KUKA KRL program: f1_Kuka_APT210T03S10.SRC

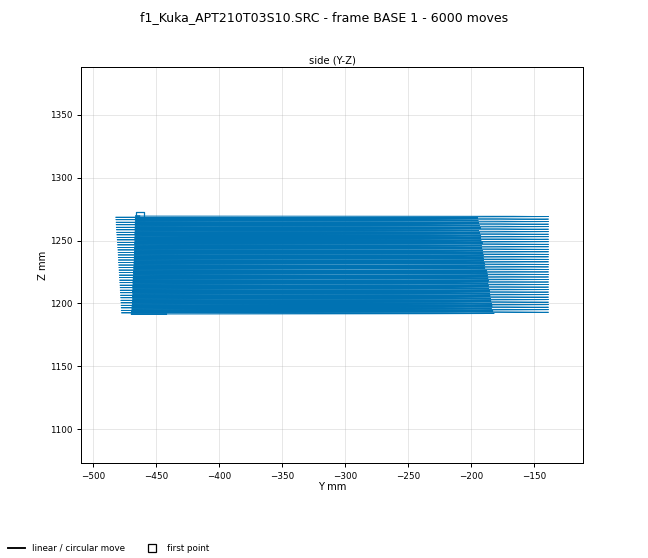
[picture p0: tool path of f1_Kuka_APT210T03S10.SRC in frame BASE 1, 6000 of 6001 moves have a stored position in this frame; points joined in program order, loops and branches not executed]
&ACCESS RVP
&REL 2
&PARAM TEMPLATE = C:\KRC\Roboter\Template\vorgabe
&PARAM EDITMASK = *
DEF f1_Kuka_APT210T03S10()


;FOLD INI;%{PE}%V3.2.0,%MKUKATPBASIS,%CINIT,%VCOMMON,%P
  ;FOLD BAS INI;%{E}%V3.2.0,%MKUKATPBASIS,%CINIT,%VINIT,%P
    GLOBAL INTERRUPT DECL 3 WHEN $STOPMESS==TRUE DO IR_STOPM ( )
    INTERRUPT ON 3
    BAS (#INITMOV,0 )
  ;ENDFOLD (BAS INI)
  ;FOLD USER INI;%{E}%V3.2.0,%MKUKATPUSER,%CINIT,%VINIT,%P
    ;Make your modifications here
  ;ENDFOLD (USER INI)
;ENDFOLD (INI)


;*** Make Null PTP Move
  PTP $pos_act

;*** Auto Load The Correct TOOL Data
  $tool=tool_data[3]

;*** Auto Load The Correct BASE Data
  $base=base_data[1]

  $ADVANCE = 5

;*** Restate Last Velocity
MMPM(30000.0)
SetRPM(6000)
LIN {X 0.158,Y -463.021,Z 1269.560,A 0.000,B 0.000,C 90.000,E1 280.725} C_DIS
LIN {X -0.171,Y -464.425,Z 1269.557,A 0.000,B 0.000,C 90.000,E1 280.254} C_DIS
LIN {X -0.038,Y -465.530,Z 1269.554,A 0.000,B 0.000,C 90.000,E1 279.726} C_DIS
LIN {X 0.024,Y -466.258,Z 1269.551,A 0.000,B 0.000,C 90.000,E1 279.208} C_DIS
LIN {X 0.098,Y -466.685,Z 1269.548,A 0.000,B 0.000,C 90.000,E1 278.690} C_DIS
LIN {X 0.243,Y -466.710,Z 1269.546,A 0.000,B 0.000,C 90.000,E1 278.163} C_DIS
LIN {X -0.138,Y -466.297,Z 1269.543,A 0.000,B 0.000,C 90.000,E1 277.701} C_DIS
LIN {X -0.055,Y -465.423,Z 1269.540,A 0.000,B 0.000,C 90.000,E1 277.182} C_DIS
LIN {X 0.026,Y -464.151,Z 1269.537,A 0.000,B 0.000,C 90.000,E1 276.663} C_DIS
LIN {X 0.102,Y -462.450,Z 1269.534,A 0.000,B 0.000,C 90.000,E1 276.144} C_DIS
LIN {X -0.010,Y -459.279,Z 1269.530,A 0.000,B 0.000,C 90.000,E1 275.391} C_DIS
LIN {X -0.004,Y -456.730,Z 1269.527,A 0.000,B 0.000,C 90.000,E1 274.878} C_DIS
LIN {X 0.028,Y -453.616,Z 1269.524,A 0.000,B 0.000,C 90.000,E1 274.359} C_DIS
LIN {X -0.204,Y -451.853,Z 1269.523,A 0.000,B 0.000,C 90.000,E1 274.131} C_DIS
LIN {X 0.039,Y -449.773,Z 1269.521,A 0.000,B 0.000,C 90.000,E1 273.841} C_DIS
LIN {X 0.001,Y -444.794,Z 1269.518,A 0.000,B 0.000,C 90.000,E1 273.326} C_DIS
LIN {X -0.204,Y -438.833,Z 1269.516,A 0.000,B 0.000,C 90.000,E1 272.865} C_DIS
LIN {X 0.074,Y -432.298,Z 1269.513,A 0.000,B 0.000,C 90.000,E1 272.407} C_DIS
LIN {X -0.016,Y -425.467,Z 1269.511,A 0.000,B 0.000,C 90.000,E1 272.064} C_DIS
LIN {X -0.063,Y -418.581,Z 1269.510,A 0.000,B 0.000,C 90.000,E1 271.776} C_DIS
LIN {X -0.186,Y -411.540,Z 1269.508,A 0.000,B 0.000,C 90.000,E1 271.547} C_DIS
LIN {X -0.025,Y -404.479,Z 1269.507,A 0.000,B 0.000,C 90.000,E1 271.318} C_DIS
LIN {X -0.034,Y -397.370,Z 1269.506,A 0.000,B 0.000,C 90.000,E1 271.146} C_DIS
LIN {X 0.152,Y -389.939,Z 1269.505,A 0.000,B 0.000,C 90.000,E1 270.974} C_DIS
LIN {X 0.139,Y -381.517,Z 1269.505,A 0.000,B 0.000,C 90.000,E1 270.859} C_DIS
LIN {X 0.169,Y -367.307,Z 1269.504,A 0.000,B 0.000,C 90.000,E1 270.745} C_DIS
LIN {X 0.045,Y -359.990,Z 1269.504,A 0.000,B 0.000,C 90.000,E1 270.745} C_DIS
LIN {X -0.008,Y -181.516,Z 1269.504,A 0.000,B 0.000,C 90.000,E1 270.745} C_DIS
LIN {X -0.022,Y -181.492,Z 1269.498,A 0.000,B 0.000,C 90.000,E1 269.714} C_DIS
LIN {X -0.079,Y -180.906,Z 1269.474,A 0.000,B 0.000,C 90.000,E1 265.355} C_DIS
LIN {X -0.005,Y -180.669,Z 1269.469,A 0.000,B 0.000,C 90.000,E1 264.489} C_DIS
LIN {X 0.070,Y -178.750,Z 1269.441,A 0.000,B 0.000,C 90.000,E1 259.398} C_DIS
LIN {X -0.033,Y -175.797,Z 1269.413,A 0.000,B 0.000,C 90.000,E1 254.338} C_DIS
LIN {X -0.038,Y -171.983,Z 1269.384,A 0.000,B 0.000,C 90.000,E1 249.209} C_DIS
LIN {X -0.001,Y -171.388,Z 1269.380,A 0.000,B 0.000,C 90.000,E1 248.337} C_DIS
LIN {X -0.015,Y -167.632,Z 1269.356,A 0.000,B 0.000,C 90.000,E1 244.024} C_DIS
LIN {X 0.000,Y -166.289,Z 1269.346,A 0.000,B 0.000,C 90.000,E1 242.281} C_DIS
LIN {X -0.006,Y -163.036,Z 1269.327,A 0.000,B 0.000,C 90.000,E1 238.791} C_DIS
LIN {X -0.044,Y -160.966,Z 1269.312,A 0.000,B 0.000,C 90.000,E1 236.167} C_DIS
LIN {X -0.066,Y -157.719,Z 1269.292,A 0.000,B 0.000,C 90.000,E1 232.637} C_DIS
LIN {X 0.092,Y -155.759,Z 1269.277,A 0.000,B 0.000,C 90.000,E1 229.908} C_DIS
LIN {X -0.071,Y -152.014,Z 1269.253,A 0.000,B 0.000,C 90.000,E1 225.486} C_DIS
LIN {X -0.053,Y -150.261,Z 1269.238,A 0.000,B 0.000,C 90.000,E1 222.771} C_DIS
LIN {X -0.034,Y -147.015,Z 1269.212,A 0.000,B 0.000,C 90.000,E1 218.222} C_DIS
LIN {X -0.013,Y -145.598,Z 1269.197,A 0.000,B 0.000,C 90.000,E1 215.471} C_DIS
LIN {X -0.009,Y -142.984,Z 1269.172,A 0.000,B 0.000,C 90.000,E1 210.875} C_DIS
LIN {X -0.009,Y -141.612,Z 1269.151,A 0.000,B 0.000,C 90.000,E1 207.180} C_DIS
LIN {X 0.032,Y -139.428,Z 1269.115,A 0.000,B 0.000,C 90.000,E1 200.663} C_DIS
LIN {X 0.083,Y -139.157,Z 1269.104,A 0.000,B 0.000,C 90.000,E1 198.779} C_DIS
LIN {X -0.031,Y -138.343,Z 1269.058,A 0.000,B 0.000,C 90.000,E1 190.423} C_DIS
LIN {X -0.049,Y -139.481,Z 1269.006,A 0.000,B 0.000,C 90.000,E1 181.088} C_DIS
LIN {X 0.031,Y -141.073,Z 1268.975,A 0.000,B 0.000,C 90.000,E1 175.469} C_DIS
LIN {X -0.014,Y -142.449,Z 1268.959,A 0.000,B 0.000,C 90.000,E1 172.704} C_DIS
LIN {X 0.076,Y -144.690,Z 1268.934,A 0.000,B 0.000,C 90.000,E1 168.049} C_DIS
LIN {X 0.028,Y -147.283,Z 1268.913,A 0.000,B 0.000,C 90.000,E1 164.393} C_DIS
LIN {X 0.045,Y -150.601,Z 1268.888,A 0.000,B 0.000,C 90.000,E1 159.826} C_DIS
LIN {X -0.019,Y -154.074,Z 1268.868,A 0.000,B 0.000,C 90.000,E1 156.230} C_DIS
LIN {X 0.047,Y -157.495,Z 1268.848,A 0.000,B 0.000,C 90.000,E1 152.615} C_DIS
LIN {X -0.008,Y -161.723,Z 1268.828,A 0.000,B 0.000,C 90.000,E1 149.076} C_DIS
LIN {X 0.006,Y -165.916,Z 1268.809,A 0.000,B 0.000,C 90.000,E1 145.548} C_DIS
LIN {X -0.008,Y -170.902,Z 1268.789,A 0.000,B 0.000,C 90.000,E1 142.065} C_DIS
LIN {X 0.019,Y -175.771,Z 1268.770,A 0.000,B 0.000,C 90.000,E1 138.609} C_DIS
LIN {X 0.020,Y -181.380,Z 1268.751,A 0.000,B 0.000,C 90.000,E1 135.202} C_DIS
LIN {X 0.025,Y -186.876,Z 1268.732,A 0.000,B 0.000,C 90.000,E1 131.838} C_DIS
LIN {X -0.023,Y -191.460,Z 1268.719,A 0.000,B 0.000,C 90.000,E1 129.358} C_DIS
LIN {X -0.091,Y -197.316,Z 1268.700,A 0.000,B 0.000,C 90.000,E1 126.091} C_DIS
LIN {X 0.035,Y -200.055,Z 1268.693,A 0.000,B 0.000,C 90.000,E1 124.692} C_DIS
LIN {X 0.012,Y -310.049,Z 1268.693,A 0.000,B 0.000,C 90.000,E1 124.692} C_DIS
LIN {X -0.114,Y -311.370,Z 1268.693,A 0.000,B 0.000,C 90.000,E1 124.692} C_DIS
LIN {X 0.173,Y -316.311,Z 1268.691,A 0.000,B 0.000,C 90.000,E1 124.405} C_DIS
LIN {X 0.136,Y -319.511,Z 1268.690,A 0.000,B 0.000,C 90.000,E1 124.119} C_DIS
LIN {X -0.031,Y -323.137,Z 1268.687,A 0.000,B 0.000,C 90.000,E1 123.627} C_DIS
LIN {X 0.048,Y -324.685,Z 1268.685,A 0.000,B 0.000,C 90.000,E1 123.293} C_DIS
LIN {X -0.059,Y -338.983,Z 1268.664,A 0.000,B 0.000,C 90.000,E1 119.539} C_DIS
LIN {X 0.108,Y -351.212,Z 1268.649,A 0.000,B 0.000,C 90.000,E1 116.744} C_DIS
LIN {X -0.164,Y -364.920,Z 1268.634,A 0.000,B 0.000,C 90.000,E1 114.079} C_DIS
LIN {X -0.132,Y -378.444,Z 1268.620,A 0.000,B 0.000,C 90.000,E1 111.716} C_DIS
LIN {X -0.031,Y -393.330,Z 1268.608,A 0.000,B 0.000,C 90.000,E1 109.396} C_DIS
LIN {X -0.067,Y -409.679,Z 1268.595,A 0.000,B 0.000,C 90.000,E1 107.149} C_DIS
LIN {X -0.068,Y -427.608,Z 1268.583,A 0.000,B 0.000,C 90.000,E1 104.954} C_DIS
LIN {X -0.038,Y -447.106,Z 1268.571,A 0.000,B 0.000,C 90.000,E1 102.827} C_DIS
LIN {X 0.166,Y -467.351,Z 1268.560,A 0.000,B 0.000,C 90.000,E1 100.838} C_DIS
LIN {X 0.180,Y -475.077,Z 1268.557,A 0.000,B 0.000,C 90.000,E1 100.141} C_DIS
LIN {X 0.231,Y -477.182,Z 1268.555,A 0.000,B 0.000,C 90.000,E1 99.905} C_DIS
LIN {X -0.191,Y -478.780,Z 1268.554,A 0.000,B 0.000,C 90.000,E1 99.726} C_DIS
LIN {X 0.075,Y -480.108,Z 1268.552,A 0.000,B 0.000,C 90.000,E1 99.443} C_DIS
LIN {X -0.053,Y -481.089,Z 1268.551,A 0.000,B 0.000,C 90.000,E1 99.208} C_DIS
LIN {X 0.108,Y -482.190,Z 1268.548,A 0.000,B 0.000,C 90.000,E1 98.690} C_DIS
LIN {X -0.131,Y -482.289,Z 1268.546,A 0.000,B 0.000,C 90.000,E1 98.219} C_DIS
LIN {X 0.042,Y -481.405,Z 1268.543,A 0.000,B 0.000,C 90.000,E1 97.701} C_DIS
LIN {X 0.217,Y -479.386,Z 1268.540,A 0.000,B 0.000,C 90.000,E1 97.182} C_DIS
LIN {X 0.093,Y -477.822,Z 1268.539,A 0.000,B 0.000,C 90.000,E1 96.947} C_DIS
LIN {X -0.096,Y -461.310,Z 1268.526,A 0.000,B 0.000,C 90.000,E1 94.702} C_DIS
LIN {X 0.147,Y -445.618,Z 1268.513,A 0.000,B 0.000,C 90.000,E1 92.350} C_DIS
LIN {X -0.178,Y -432.570,Z 1268.501,A 0.000,B 0.000,C 90.000,E1 90.286} C_DIS
LIN {X 0.076,Y -414.803,Z 1268.484,A 0.000,B 0.000,C 90.000,E1 87.020} C_DIS
LIN {X -0.112,Y -404.774,Z 1268.473,A 0.000,B 0.000,C 90.000,E1 85.122} C_DIS
LIN {X -0.122,Y -396.062,Z 1268.464,A 0.000,B 0.000,C 90.000,E1 83.451} C_DIS
LIN {X 0.134,Y -385.703,Z 1268.453,A 0.000,B 0.000,C 90.000,E1 81.432} C_DIS
LIN {X -0.114,Y -376.640,Z 1268.443,A 0.000,B 0.000,C 90.000,E1 79.746} C_DIS
LIN {X -0.080,Y -367.188,Z 1268.433,A 0.000,B 0.000,C 90.000,E1 77.993} C_DIS
LIN {X -0.100,Y -359.050,Z 1268.425,A 0.000,B 0.000,C 90.000,E1 76.520} C_DIS
LIN {X 0.054,Y -347.571,Z 1268.413,A 0.000,B 0.000,C 90.000,E1 74.393} C_DIS
LIN {X 0.032,Y -334.469,Z 1268.400,A 0.000,B 0.000,C 90.000,E1 71.945} C_DIS
LIN {X -0.036,Y -320.293,Z 1268.384,A 0.000,B 0.000,C 90.000,E1 69.135} C_DIS
LIN {X -0.150,Y -304.085,Z 1268.364,A 0.000,B 0.000,C 90.000,E1 65.613} C_DIS
LIN {X -0.020,Y -292.232,Z 1268.348,A 0.000,B 0.000,C 90.000,E1 62.615} C_DIS
LIN {X 0.106,Y -279.452,Z 1268.327,A 0.000,B 0.000,C 90.000,E1 58.869} C_DIS
LIN {X -0.065,Y -270.033,Z 1268.310,A 0.000,B 0.000,C 90.000,E1 55.801} C_DIS
LIN {X 0.025,Y -260.411,Z 1268.290,A 0.000,B 0.000,C 90.000,E1 52.271} C_DIS
LIN {X 0.015,Y -253.234,Z 1268.275,A 0.000,B 0.000,C 90.000,E1 49.417} C_DIS
LIN {X -0.068,Y -244.624,Z 1268.254,A 0.000,B 0.000,C 90.000,E1 45.810} C_DIS
LIN {X -0.071,Y -236.646,Z 1268.234,A 0.000,B 0.000,C 90.000,E1 42.123} C_DIS
LIN {X -0.096,Y -229.157,Z 1268.213,A 0.000,B 0.000,C 90.000,E1 38.382} C_DIS
LIN {X 0.083,Y -222.331,Z 1268.192,A 0.000,B 0.000,C 90.000,E1 34.532} C_DIS
LIN {X 0.099,Y -216.238,Z 1268.171,A 0.000,B 0.000,C 90.000,E1 30.669} C_DIS
LIN {X -0.029,Y -210.768,Z 1268.149,A 0.000,B 0.000,C 90.000,E1 26.796} C_DIS
LIN {X 0.046,Y -206.032,Z 1268.127,A 0.000,B 0.000,C 90.000,E1 22.823} C_DIS
LIN {X -0.048,Y -201.303,Z 1268.100,A 0.000,B 0.000,C 90.000,E1 18.055} C_DIS
LIN {X 0.084,Y -197.587,Z 1268.073,A 0.000,B 0.000,C 90.000,E1 13.175} C_DIS
LIN {X -0.088,Y -194.592,Z 1268.042,A 0.000,B 0.000,C 90.000,E1 7.530} C_DIS
LIN {X -0.068,Y -195.631,Z 1267.956,A 0.000,B 0.000,C 90.000,E1 352.186} C_DIS
LIN {X 0.023,Y -199.328,Z 1267.925,A 0.000,B 0.000,C 90.000,E1 346.464} C_DIS
LIN {X -0.029,Y -203.599,Z 1267.898,A 0.000,B 0.000,C 90.000,E1 341.638} C_DIS
LIN {X 0.062,Y -207.896,Z 1267.876,A 0.000,B 0.000,C 90.000,E1 337.614} C_DIS
LIN {X 0.115,Y -212.948,Z 1267.854,A 0.000,B 0.000,C 90.000,E1 333.640} C_DIS
LIN {X 0.043,Y -218.627,Z 1267.832,A 0.000,B 0.000,C 90.000,E1 329.744} C_DIS
LIN {X 0.023,Y -225.096,Z 1267.810,A 0.000,B 0.000,C 90.000,E1 325.881} C_DIS
LIN {X 0.029,Y -232.402,Z 1267.789,A 0.000,B 0.000,C 90.000,E1 322.065} C_DIS
LIN {X -0.034,Y -240.571,Z 1267.768,A 0.000,B 0.000,C 90.000,E1 318.324} C_DIS
LIN {X 0.122,Y -249.787,Z 1267.748,A 0.000,B 0.000,C 90.000,E1 314.595} C_DIS
LIN {X 0.007,Y -257.116,Z 1267.734,A 0.000,B 0.000,C 90.000,E1 312.081} C_DIS
LIN {X 0.077,Y -265.464,Z 1267.720,A 0.000,B 0.000,C 90.000,E1 309.564} C_DIS
LIN {X 0.122,Y -273.667,Z 1267.708,A 0.000,B 0.000,C 90.000,E1 307.443} C_DIS
LIN {X -0.005,Y -282.937,Z 1267.697,A 0.000,B 0.000,C 90.000,E1 305.391} C_DIS
LIN {X -0.123,Y -293.218,Z 1267.685,A 0.000,B 0.000,C 90.000,E1 303.372} C_DIS
LIN {X 0.028,Y -302.560,Z 1267.676,A 0.000,B 0.000,C 90.000,E1 301.671} C_DIS
LIN {X 0.134,Y -310.858,Z 1267.669,A 0.000,B 0.000,C 90.000,E1 300.335} C_DIS
LIN {X -0.082,Y -319.939,Z 1267.661,A 0.000,B 0.000,C 90.000,E1 299.077} C_DIS
LIN {X -0.060,Y -339.665,Z 1267.647,A 0.000,B 0.000,C 90.000,E1 296.539} C_DIS
LIN {X 0.032,Y -357.895,Z 1267.635,A 0.000,B 0.000,C 90.000,E1 294.387} C_DIS
LIN {X 0.075,Y -370.867,Z 1267.627,A 0.000,B 0.000,C 90.000,E1 292.898} C_DIS
LIN {X -0.027,Y -383.639,Z 1267.619,A 0.000,B 0.000,C 90.000,E1 291.461} C_DIS
LIN {X -0.057,Y -398.664,Z 1267.610,A 0.000,B 0.000,C 90.000,E1 289.758} C_DIS
LIN {X -0.116,Y -416.277,Z 1267.599,A 0.000,B 0.000,C 90.000,E1 287.873} C_DIS
LIN {X -0.219,Y -426.089,Z 1267.593,A 0.000,B 0.000,C 90.000,E1 286.804} C_DIS
LIN {X -0.040,Y -432.978,Z 1267.589,A 0.000,B 0.000,C 90.000,E1 285.969} C_DIS
LIN {X -0.210,Y -439.391,Z 1267.584,A 0.000,B 0.000,C 90.000,E1 285.190} C_DIS
LIN {X 0.092,Y -445.134,Z 1267.580,A 0.000,B 0.000,C 90.000,E1 284.356} C_DIS
LIN {X -0.088,Y -450.216,Z 1267.575,A 0.000,B 0.000,C 90.000,E1 283.592} C_DIS
LIN {X -0.229,Y -454.646,Z 1267.571,A 0.000,B 0.000,C 90.000,E1 282.827} C_DIS
LIN {X 0.120,Y -458.319,Z 1267.567,A 0.000,B 0.000,C 90.000,E1 282.007} C_DIS
LIN {X 0.052,Y -461.356,Z 1267.563,A 0.000,B 0.000,C 90.000,E1 281.243} C_DIS
LIN {X 0.079,Y -463.002,Z 1267.560,A 0.000,B 0.000,C 90.000,E1 280.725} C_DIS
LIN {X 0.206,Y -464.426,Z 1267.557,A 0.000,B 0.000,C 90.000,E1 280.197} C_DIS
LIN {X -0.119,Y -465.517,Z 1267.554,A 0.000,B 0.000,C 90.000,E1 279.726} C_DIS
LIN {X -0.057,Y -466.289,Z 1267.551,A 0.000,B 0.000,C 90.000,E1 279.208} C_DIS
LIN {X 0.087,Y -466.729,Z 1267.548,A 0.000,B 0.000,C 90.000,E1 278.681} C_DIS
LIN {X 0.163,Y -466.768,Z 1267.545,A 0.000,B 0.000,C 90.000,E1 278.163} C_DIS
LIN {X -0.218,Y -466.373,Z 1267.543,A 0.000,B 0.000,C 90.000,E1 277.701} C_DIS
LIN {X -0.135,Y -465.526,Z 1267.540,A 0.000,B 0.000,C 90.000,E1 277.182} C_DIS
LIN {X -0.053,Y -464.254,Z 1267.537,A 0.000,B 0.000,C 90.000,E1 276.663} C_DIS
LIN {X 0.023,Y -462.607,Z 1267.534,A 0.000,B 0.000,C 90.000,E1 276.144} C_DIS
LIN {X -0.086,Y -459.480,Z 1267.530,A 0.000,B 0.000,C 90.000,E1 275.391} C_DIS
LIN {X -0.078,Y -456.957,Z 1267.527,A 0.000,B 0.000,C 90.000,E1 274.878} C_DIS
LIN {X -0.046,Y -453.897,Z 1267.524,A 0.000,B 0.000,C 90.000,E1 274.359} C_DIS
LIN {X -0.033,Y -450.045,Z 1267.521,A 0.000,B 0.000,C 90.000,E1 273.841} C_DIS
LIN {X -0.068,Y -445.071,Z 1267.518,A 0.000,B 0.000,C 90.000,E1 273.326} C_DIS
LIN {X 0.140,Y -439.130,Z 1267.516,A 0.000,B 0.000,C 90.000,E1 272.808} C_DIS
LIN {X -0.049,Y -432.570,Z 1267.513,A 0.000,B 0.000,C 90.000,E1 272.407} C_DIS
LIN {X -0.148,Y -425.696,Z 1267.511,A 0.000,B 0.000,C 90.000,E1 272.064} C_DIS
LIN {X 0.202,Y -418.795,Z 1267.510,A 0.000,B 0.000,C 90.000,E1 271.718} C_DIS
LIN {X 0.061,Y -411.685,Z 1267.508,A 0.000,B 0.000,C 90.000,E1 271.489} C_DIS
LIN {X -0.045,Y -400.883,Z 1267.507,A 0.000,B 0.000,C 90.000,E1 271.203} C_DIS
LIN {X -0.026,Y -389.864,Z 1267.505,A 0.000,B 0.000,C 90.000,E1 270.974} C_DIS
LIN {X -0.034,Y -381.152,Z 1267.505,A 0.000,B 0.000,C 90.000,E1 270.859} C_DIS
LIN {X 0.002,Y -366.340,Z 1267.504,A 0.000,B 0.000,C 90.000,E1 270.745} C_DIS
LIN {X -0.060,Y -363.755,Z 1267.504,A 0.000,B 0.000,C 90.000,E1 270.745} C_DIS
LIN {X -0.062,Y -181.520,Z 1267.504,A 0.000,B 0.000,C 90.000,E1 270.745} C_DIS
LIN {X -0.014,Y -181.493,Z 1267.498,A 0.000,B 0.000,C 90.000,E1 269.714} C_DIS
LIN {X -0.071,Y -180.905,Z 1267.474,A 0.000,B 0.000,C 90.000,E1 265.355} C_DIS
LIN {X 0.003,Y -180.670,Z 1267.469,A 0.000,B 0.000,C 90.000,E1 264.489} C_DIS
LIN {X 0.077,Y -178.751,Z 1267.441,A 0.000,B 0.000,C 90.000,E1 259.398} C_DIS
LIN {X -0.026,Y -175.799,Z 1267.413,A 0.000,B 0.000,C 90.000,E1 254.338} C_DIS
LIN {X -0.030,Y -171.984,Z 1267.384,A 0.000,B 0.000,C 90.000,E1 249.209} C_DIS
LIN {X 0.008,Y -171.390,Z 1267.380,A 0.000,B 0.000,C 90.000,E1 248.337} C_DIS
LIN {X -0.008,Y -167.634,Z 1267.356,A 0.000,B 0.000,C 90.000,E1 244.024} C_DIS
LIN {X 0.008,Y -166.291,Z 1267.346,A 0.000,B 0.000,C 90.000,E1 242.281} C_DIS
LIN {X 0.002,Y -163.038,Z 1267.327,A 0.000,B 0.000,C 90.000,E1 238.791} C_DIS
LIN {X -0.037,Y -160.969,Z 1267.312,A 0.000,B 0.000,C 90.000,E1 236.167} C_DIS
LIN {X -0.059,Y -157.721,Z 1267.292,A 0.000,B 0.000,C 90.000,E1 232.637} C_DIS
LIN {X 0.100,Y -155.760,Z 1267.277,A 0.000,B 0.000,C 90.000,E1 229.908} C_DIS
LIN {X -0.063,Y -152.017,Z 1267.253,A 0.000,B 0.000,C 90.000,E1 225.486} C_DIS
LIN {X -0.045,Y -150.263,Z 1267.238,A 0.000,B 0.000,C 90.000,E1 222.771} C_DIS
LIN {X -0.027,Y -147.017,Z 1267.212,A 0.000,B 0.000,C 90.000,E1 218.222} C_DIS
LIN {X -0.006,Y -145.599,Z 1267.197,A 0.000,B 0.000,C 90.000,E1 215.471} C_DIS
LIN {X -0.002,Y -142.986,Z 1267.172,A 0.000,B 0.000,C 90.000,E1 210.875} C_DIS
LIN {X -0.002,Y -141.613,Z 1267.151,A 0.000,B 0.000,C 90.000,E1 207.180} C_DIS
LIN {X 0.039,Y -139.428,Z 1267.115,A 0.000,B 0.000,C 90.000,E1 200.663} C_DIS
LIN {X -0.042,Y -139.158,Z 1267.104,A 0.000,B 0.000,C 90.000,E1 198.833} C_DIS
LIN {X -0.024,Y -138.342,Z 1267.058,A 0.000,B 0.000,C 90.000,E1 190.423} C_DIS
LIN {X -0.042,Y -139.481,Z 1267.006,A 0.000,B 0.000,C 90.000,E1 181.088} C_DIS
LIN {X 0.039,Y -141.073,Z 1266.975,A 0.000,B 0.000,C 90.000,E1 175.469} C_DIS
LIN {X -0.007,Y -142.448,Z 1266.959,A 0.000,B 0.000,C 90.000,E1 172.704} C_DIS
LIN {X 0.083,Y -144.689,Z 1266.934,A 0.000,B 0.000,C 90.000,E1 168.049} C_DIS
LIN {X 0.036,Y -147.281,Z 1266.913,A 0.000,B 0.000,C 90.000,E1 164.393} C_DIS
LIN {X 0.052,Y -150.599,Z 1266.888,A 0.000,B 0.000,C 90.000,E1 159.826} C_DIS
LIN {X -0.012,Y -154.072,Z 1266.868,A 0.000,B 0.000,C 90.000,E1 156.230} C_DIS
LIN {X 0.054,Y -157.492,Z 1266.848,A 0.000,B 0.000,C 90.000,E1 152.615} C_DIS
LIN {X 0.000,Y -161.719,Z 1266.828,A 0.000,B 0.000,C 90.000,E1 149.076} C_DIS
LIN {X 0.013,Y -165.913,Z 1266.809,A 0.000,B 0.000,C 90.000,E1 145.548} C_DIS
LIN {X 0.001,Y -170.899,Z 1266.789,A 0.000,B 0.000,C 90.000,E1 142.065} C_DIS
LIN {X 0.028,Y -175.767,Z 1266.770,A 0.000,B 0.000,C 90.000,E1 138.609} C_DIS
LIN {X -0.100,Y -181.376,Z 1266.751,A 0.000,B 0.000,C 90.000,E1 135.243} C_DIS
LIN {X 0.033,Y -186.871,Z 1266.733,A 0.000,B 0.000,C 90.000,E1 131.838} C_DIS
LIN {X -0.014,Y -191.455,Z 1266.719,A 0.000,B 0.000,C 90.000,E1 129.358} C_DIS
LIN {X -0.082,Y -197.310,Z 1266.700,A 0.000,B 0.000,C 90.000,E1 126.091} C_DIS
LIN {X -0.012,Y -200.083,Z 1266.693,A 0.000,B 0.000,C 90.000,E1 124.692} C_DIS
LIN {X -0.061,Y -309.766,Z 1266.693,A 0.000,B 0.000,C 90.000,E1 124.692} C_DIS
LIN {X -0.073,Y -316.076,Z 1266.691,A 0.000,B 0.000,C 90.000,E1 124.452} C_DIS
LIN {X -0.096,Y -319.047,Z 1266.690,A 0.000,B 0.000,C 90.000,E1 124.199} C_DIS
LIN {X -0.141,Y -322.741,Z 1266.687,A 0.000,B 0.000,C 90.000,E1 123.706} C_DIS
LIN {X -0.063,Y -324.386,Z 1266.685,A 0.000,B 0.000,C 90.000,E1 123.372} C_DIS
LIN {X -0.062,Y -327.900,Z 1266.680,A 0.000,B 0.000,C 90.000,E1 122.418} C_DIS
LIN {X -0.010,Y -338.723,Z 1266.664,A 0.000,B 0.000,C 90.000,E1 119.589} C_DIS
LIN {X -0.016,Y -350.922,Z 1266.649,A 0.000,B 0.000,C 90.000,E1 116.821} C_DIS
LIN {X 0.189,Y -364.596,Z 1266.634,A 0.000,B 0.000,C 90.000,E1 114.079} C_DIS
LIN {X -0.125,Y -378.092,Z 1266.621,A 0.000,B 0.000,C 90.000,E1 111.770} C_DIS
LIN {X -0.039,Y -392.943,Z 1266.608,A 0.000,B 0.000,C 90.000,E1 109.450} C_DIS
LIN {X -0.212,Y -409.258,Z 1266.595,A 0.000,B 0.000,C 90.000,E1 107.221} C_DIS
LIN {X -0.107,Y -427.148,Z 1266.583,A 0.000,B 0.000,C 90.000,E1 105.009} C_DIS
LIN {X -0.102,Y -446.616,Z 1266.572,A 0.000,B 0.000,C 90.000,E1 102.883} C_DIS
LIN {X 0.063,Y -466.847,Z 1266.561,A 0.000,B 0.000,C 90.000,E1 100.894} C_DIS
LIN {X 0.062,Y -474.584,Z 1266.557,A 0.000,B 0.000,C 90.000,E1 100.197} C_DIS
LIN {X 0.117,Y -476.776,Z 1266.555,A 0.000,B 0.000,C 90.000,E1 99.962} C_DIS
LIN {X 0.170,Y -478.434,Z 1266.554,A 0.000,B 0.000,C 90.000,E1 99.726} C_DIS
LIN {X -0.038,Y -479.815,Z 1266.553,A 0.000,B 0.000,C 90.000,E1 99.500} C_DIS
LIN {X -0.167,Y -480.839,Z 1266.551,A 0.000,B 0.000,C 90.000,E1 99.265} C_DIS
LIN {X -0.010,Y -482.013,Z 1266.549,A 0.000,B 0.000,C 90.000,E1 98.746} C_DIS
LIN {X 0.227,Y -482.176,Z 1266.546,A 0.000,B 0.000,C 90.000,E1 98.219} C_DIS
LIN {X -0.078,Y -481.361,Z 1266.543,A 0.000,B 0.000,C 90.000,E1 97.757} C_DIS
LIN {X 0.095,Y -479.428,Z 1266.540,A 0.000,B 0.000,C 90.000,E1 97.239} C_DIS
LIN {X -0.029,Y -477.924,Z 1266.539,A 0.000,B 0.000,C 90.000,E1 97.004} C_DIS
LIN {X 0.029,Y -459.641,Z 1266.525,A 0.000,B 0.000,C 90.000,E1 94.473} C_DIS
LIN {X -0.209,Y -444.016,Z 1266.512,A 0.000,B 0.000,C 90.000,E1 92.178} C_DIS
LIN {X 0.149,Y -432.605,Z 1266.502,A 0.000,B 0.000,C 90.000,E1 90.286} C_DIS
LIN {X -0.120,Y -416.277,Z 1266.485,A 0.000,B 0.000,C 90.000,E1 87.364} C_DIS
LIN {X 0.196,Y -404.829,Z 1266.473,A 0.000,B 0.000,C 90.000,E1 85.122} C_DIS
LIN {X 0.135,Y -396.116,Z 1266.464,A 0.000,B 0.000,C 90.000,E1 83.457} C_DIS
LIN {X 0.048,Y -385.759,Z 1266.453,A 0.000,B 0.000,C 90.000,E1 81.489} C_DIS
LIN {X 0.175,Y -376.705,Z 1266.443,A 0.000,B 0.000,C 90.000,E1 79.746} C_DIS
LIN {X -0.157,Y -367.282,Z 1266.433,A 0.000,B 0.000,C 90.000,E1 78.049} C_DIS
LIN {X 0.138,Y -357.506,Z 1266.424,A 0.000,B 0.000,C 90.000,E1 76.228} C_DIS
LIN {X -0.080,Y -346.034,Z 1266.412,A 0.000,B 0.000,C 90.000,E1 74.157} C_DIS
LIN {X -0.033,Y -332.990,Z 1266.398,A 0.000,B 0.000,C 90.000,E1 71.692} C_DIS
LIN {X 0.050,Y -318.884,Z 1266.383,A 0.000,B 0.000,C 90.000,E1 68.847} C_DIS
LIN {X -0.002,Y -302.828,Z 1266.363,A 0.000,B 0.000,C 90.000,E1 65.305} C_DIS
LIN {X -0.179,Y -291.108,Z 1266.346,A 0.000,B 0.000,C 90.000,E1 62.359} C_DIS
LIN {X -0.083,Y -278.399,Z 1266.326,A 0.000,B 0.000,C 90.000,E1 58.614} C_DIS
LIN {X 0.018,Y -268.019,Z 1266.306,A 0.000,B 0.000,C 90.000,E1 55.135} C_DIS
LIN {X -0.015,Y -258.521,Z 1266.287,A 0.000,B 0.000,C 90.000,E1 51.618} C_DIS
LIN {X -0.101,Y -251.379,Z 1266.271,A 0.000,B 0.000,C 90.000,E1 48.771} C_DIS
LIN {X 0.115,Y -242.871,Z 1266.251,A 0.000,B 0.000,C 90.000,E1 45.081} C_DIS
LIN {X -0.040,Y -236.536,Z 1266.234,A 0.000,B 0.000,C 90.000,E1 42.162} C_DIS
LIN {X 0.084,Y -228.992,Z 1266.213,A 0.000,B 0.000,C 90.000,E1 38.382} C_DIS
LIN {X -0.056,Y -222.126,Z 1266.192,A 0.000,B 0.000,C 90.000,E1 34.612} C_DIS
LIN {X 0.071,Y -215.931,Z 1266.171,A 0.000,B 0.000,C 90.000,E1 30.718} C_DIS
LIN {X 0.021,Y -210.428,Z 1266.149,A 0.000,B 0.000,C 90.000,E1 26.821} C_DIS
LIN {X -0.092,Y -205.670,Z 1266.127,A 0.000,B 0.000,C 90.000,E1 22.898} C_DIS
LIN {X 0.067,Y -200.912,Z 1266.100,A 0.000,B 0.000,C 90.000,E1 18.055} C_DIS
LIN {X -0.055,Y -197.201,Z 1266.073,A 0.000,B 0.000,C 90.000,E1 13.244} C_DIS
LIN {X -0.008,Y -194.235,Z 1266.042,A 0.000,B 0.000,C 90.000,E1 7.530} C_DIS
LIN {X -0.081,Y -195.435,Z 1265.956,A 0.000,B 0.000,C 90.000,E1 352.186} C_DIS
LIN {X 0.001,Y -199.169,Z 1265.925,A 0.000,B 0.000,C 90.000,E1 346.464} C_DIS
LIN {X -0.057,Y -203.482,Z 1265.898,A 0.000,B 0.000,C 90.000,E1 341.638} C_DIS
LIN {X 0.031,Y -207.817,Z 1265.876,A 0.000,B 0.000,C 90.000,E1 337.614} C_DIS
LIN {X 0.080,Y -212.892,Z 1265.854,A 0.000,B 0.000,C 90.000,E1 333.640} C_DIS
LIN {X 0.005,Y -218.568,Z 1265.832,A 0.000,B 0.000,C 90.000,E1 329.744} C_DIS
LIN {X -0.018,Y -225.073,Z 1265.810,A 0.000,B 0.000,C 90.000,E1 325.881} C_DIS
LIN {X -0.014,Y -232.373,Z 1265.789,A 0.000,B 0.000,C 90.000,E1 322.065} C_DIS
LIN {X -0.080,Y -240.543,Z 1265.768,A 0.000,B 0.000,C 90.000,E1 318.324} C_DIS
LIN {X 0.073,Y -249.757,Z 1265.748,A 0.000,B 0.000,C 90.000,E1 314.595} C_DIS
LIN {X -0.043,Y -257.088,Z 1265.734,A 0.000,B 0.000,C 90.000,E1 312.081} C_DIS
LIN {X 0.025,Y -265.425,Z 1265.720,A 0.000,B 0.000,C 90.000,E1 309.564} C_DIS
LIN {X -0.010,Y -275.069,Z 1265.706,A 0.000,B 0.000,C 90.000,E1 307.111} C_DIS
LIN {X 0.055,Y -284.540,Z 1265.695,A 0.000,B 0.000,C 90.000,E1 305.025} C_DIS
LIN {X -0.035,Y -294.944,Z 1265.683,A 0.000,B 0.000,C 90.000,E1 303.007} C_DIS
LIN {X -0.023,Y -304.456,Z 1265.674,A 0.000,B 0.000,C 90.000,E1 301.337} C_DIS
LIN {X 0.159,Y -315.221,Z 1265.665,A 0.000,B 0.000,C 90.000,E1 299.667} C_DIS
LIN {X 0.069,Y -334.565,Z 1265.651,A 0.000,B 0.000,C 90.000,E1 297.129} C_DIS
LIN {X 0.034,Y -354.844,Z 1265.637,A 0.000,B 0.000,C 90.000,E1 294.719} C_DIS
LIN {X 0.152,Y -367.931,Z 1265.629,A 0.000,B 0.000,C 90.000,E1 293.206} C_DIS
LIN {X 0.015,Y -380.718,Z 1265.621,A 0.000,B 0.000,C 90.000,E1 291.770} C_DIS
LIN {X -0.028,Y -395.809,Z 1265.611,A 0.000,B 0.000,C 90.000,E1 290.066} C_DIS
LIN {X 0.040,Y -416.031,Z 1265.599,A 0.000,B 0.000,C 90.000,E1 287.873} C_DIS
LIN {X -0.053,Y -425.865,Z 1265.593,A 0.000,B 0.000,C 90.000,E1 286.804} C_DIS
LIN {X 0.125,Y -432.793,Z 1265.589,A 0.000,B 0.000,C 90.000,E1 285.969} C_DIS
LIN {X -0.044,Y -439.200,Z 1265.584,A 0.000,B 0.000,C 90.000,E1 285.190} C_DIS
LIN {X -0.172,Y -444.974,Z 1265.580,A 0.000,B 0.000,C 90.000,E1 284.411} C_DIS
LIN {X 0.080,Y -450.085,Z 1265.576,A 0.000,B 0.000,C 90.000,E1 283.592} C_DIS
LIN {X -0.061,Y -454.490,Z 1265.571,A 0.000,B 0.000,C 90.000,E1 282.827} C_DIS
LIN {X -0.160,Y -458.186,Z 1265.567,A 0.000,B 0.000,C 90.000,E1 282.063} C_DIS
LIN {X 0.219,Y -461.264,Z 1265.563,A 0.000,B 0.000,C 90.000,E1 281.243} C_DIS
LIN {X -0.209,Y -462.922,Z 1265.560,A 0.000,B 0.000,C 90.000,E1 280.782} C_DIS
LIN {X -0.084,Y -464.330,Z 1265.557,A 0.000,B 0.000,C 90.000,E1 280.254} C_DIS
LIN {X 0.048,Y -465.445,Z 1265.554,A 0.000,B 0.000,C 90.000,E1 279.726} C_DIS
LIN {X 0.111,Y -466.298,Z 1265.551,A 0.000,B 0.000,C 90.000,E1 279.208} C_DIS
LIN {X 0.183,Y -466.746,Z 1265.548,A 0.000,B 0.000,C 90.000,E1 278.690} C_DIS
LIN {X -0.132,Y -466.824,Z 1265.546,A 0.000,B 0.000,C 90.000,E1 278.219} C_DIS
LIN {X -0.051,Y -466.498,Z 1265.543,A 0.000,B 0.000,C 90.000,E1 277.701} C_DIS
LIN {X 0.032,Y -465.680,Z 1265.540,A 0.000,B 0.000,C 90.000,E1 277.182} C_DIS
LIN {X 0.114,Y -464.471,Z 1265.537,A 0.000,B 0.000,C 90.000,E1 276.663} C_DIS
LIN {X 0.191,Y -462.850,Z 1265.534,A 0.000,B 0.000,C 90.000,E1 276.144} C_DIS
LIN {X 0.082,Y -459.799,Z 1265.530,A 0.000,B 0.000,C 90.000,E1 275.391} C_DIS
LIN {X 0.091,Y -457.330,Z 1265.527,A 0.000,B 0.000,C 90.000,E1 274.878} C_DIS
LIN {X 0.123,Y -454.306,Z 1265.524,A 0.000,B 0.000,C 90.000,E1 274.359} C_DIS
LIN {X -0.106,Y -452.554,Z 1265.523,A 0.000,B 0.000,C 90.000,E1 274.131} C_DIS
LIN {X -0.098,Y -448.264,Z 1265.520,A 0.000,B 0.000,C 90.000,E1 273.612} C_DIS
LIN {X 0.103,Y -445.689,Z 1265.519,A 0.000,B 0.000,C 90.000,E1 273.326} C_DIS
LIN {X -0.156,Y -439.827,Z 1265.516,A 0.000,B 0.000,C 90.000,E1 272.865} C_DIS
LIN {X 0.046,Y -433.328,Z 1265.513,A 0.000,B 0.000,C 90.000,E1 272.407} C_DIS
LIN {X -0.097,Y -426.481,Z 1265.511,A 0.000,B 0.000,C 90.000,E1 272.064} C_DIS
LIN {X -0.199,Y -419.529,Z 1265.510,A 0.000,B 0.000,C 90.000,E1 271.776} C_DIS
LIN {X 0.055,Y -412.463,Z 1265.508,A 0.000,B 0.000,C 90.000,E1 271.489} C_DIS
LIN {X -0.100,Y -401.739,Z 1265.507,A 0.000,B 0.000,C 90.000,E1 271.203} C_DIS
LIN {X -0.087,Y -393.911,Z 1265.506,A 0.000,B 0.000,C 90.000,E1 271.031} C_DIS
LIN {X 0.174,Y -385.825,Z 1265.505,A 0.000,B 0.000,C 90.000,E1 270.859} C_DIS
LIN {X -0.135,Y -375.921,Z 1265.504,A 0.000,B 0.000,C 90.000,E1 270.802} C_DIS
LIN {X 0.152,Y -362.858,Z 1265.504,A 0.000,B 0.000,C 90.000,E1 270.688} C_DIS
LIN {X 0.044,Y -181.526,Z 1265.504,A 0.000,B 0.000,C 90.000,E1 270.688} C_DIS
LIN {X -0.090,Y -181.487,Z 1265.498,A 0.000,B 0.000,C 90.000,E1 269.714} C_DIS
LIN {X 0.034,Y -180.904,Z 1265.474,A 0.000,B 0.000,C 90.000,E1 265.298} C_DIS
LIN {X -0.016,Y -180.248,Z 1265.465,A 0.000,B 0.000,C 90.000,E1 263.628} C_DIS
LIN {X 0.002,Y -178.737,Z 1265.441,A 0.000,B 0.000,C 90.000,E1 259.398} C_DIS
LIN {X 0.069,Y -175.785,Z 1265.413,A 0.000,B 0.000,C 90.000,E1 254.283} C_DIS
LIN {X 0.056,Y -171.969,Z 1265.384,A 0.000,B 0.000,C 90.000,E1 249.156} C_DIS
LIN {X 0.094,Y -171.369,Z 1265.380,A 0.000,B 0.000,C 90.000,E1 248.284} C_DIS
LIN {X -0.080,Y -167.616,Z 1265.356,A 0.000,B 0.000,C 90.000,E1 244.024} C_DIS
LIN {X -0.065,Y -166.265,Z 1265.346,A 0.000,B 0.000,C 90.000,E1 242.281} C_DIS
LIN {X 0.070,Y -163.018,Z 1265.327,A 0.000,B 0.000,C 90.000,E1 238.742} C_DIS
LIN {X -0.017,Y -160.943,Z 1265.312,A 0.000,B 0.000,C 90.000,E1 236.135} C_DIS
LIN {X 0.093,Y -157.701,Z 1265.292,A 0.000,B 0.000,C 90.000,E1 232.557} C_DIS
LIN {X 0.031,Y -155.740,Z 1265.277,A 0.000,B 0.000,C 90.000,E1 229.908} C_DIS
LIN {X 0.084,Y -151.998,Z 1265.252,A 0.000,B 0.000,C 90.000,E1 225.405} C_DIS
LIN {X -0.010,Y -150.243,Z 1265.237,A 0.000,B 0.000,C 90.000,E1 222.732} C_DIS
LIN {X 0.022,Y -147.002,Z 1265.212,A 0.000,B 0.000,C 90.000,E1 218.177} C_DIS
LIN {X 0.012,Y -145.586,Z 1265.197,A 0.000,B 0.000,C 90.000,E1 215.438} C_DIS
LIN {X 0.006,Y -142.974,Z 1265.171,A 0.000,B 0.000,C 90.000,E1 210.846} C_DIS
LIN {X 0.059,Y -141.601,Z 1265.151,A 0.000,B 0.000,C 90.000,E1 207.129} C_DIS
LIN {X -0.026,Y -139.423,Z 1265.115,A 0.000,B 0.000,C 90.000,E1 200.663} C_DIS
LIN {X 0.026,Y -139.152,Z 1265.104,A 0.000,B 0.000,C 90.000,E1 198.779} C_DIS
LIN {X 0.048,Y -138.345,Z 1265.058,A 0.000,B 0.000,C 90.000,E1 190.366} C_DIS
LIN {X 0.033,Y -139.485,Z 1265.006,A 0.000,B 0.000,C 90.000,E1 181.031} C_DIS
LIN {X -0.026,Y -141.084,Z 1264.975,A 0.000,B 0.000,C 90.000,E1 175.469} C_DIS
LIN {X -0.073,Y -142.461,Z 1264.959,A 0.000,B 0.000,C 90.000,E1 172.704} C_DIS
LIN {X 0.017,Y -144.704,Z 1264.934,A 0.000,B 0.000,C 90.000,E1 168.049} C_DIS
LIN {X -0.032,Y -147.302,Z 1264.913,A 0.000,B 0.000,C 90.000,E1 164.393} C_DIS
LIN {X -0.016,Y -150.621,Z 1264.888,A 0.000,B 0.000,C 90.000,E1 159.826} C_DIS
LIN {X 0.060,Y -154.096,Z 1264.868,A 0.000,B 0.000,C 90.000,E1 156.177} C_DIS
LIN {X -0.016,Y -157.520,Z 1264.848,A 0.000,B 0.000,C 90.000,E1 152.615} C_DIS
LIN {X -0.071,Y -161.752,Z 1264.828,A 0.000,B 0.000,C 90.000,E1 149.076} C_DIS
LIN {X 0.034,Y -165.945,Z 1264.808,A 0.000,B 0.000,C 90.000,E1 145.515} C_DIS
LIN {X 0.032,Y -170.936,Z 1264.789,A 0.000,B 0.000,C 90.000,E1 142.029} C_DIS
LIN {X -0.048,Y -175.804,Z 1264.770,A 0.000,B 0.000,C 90.000,E1 138.609} C_DIS
LIN {X 0.080,Y -181.413,Z 1264.751,A 0.000,B 0.000,C 90.000,E1 135.162} C_DIS
LIN {X -0.045,Y -186.914,Z 1264.732,A 0.000,B 0.000,C 90.000,E1 131.838} C_DIS
LIN {X 0.028,Y -191.494,Z 1264.719,A 0.000,B 0.000,C 90.000,E1 129.322} C_DIS
LIN {X 0.114,Y -197.356,Z 1264.700,A 0.000,B 0.000,C 90.000,E1 126.011} C_DIS
LIN {X -0.065,Y -200.115,Z 1264.693,A 0.000,B 0.000,C 90.000,E1 124.692} C_DIS
LIN {X -0.143,Y -309.647,Z 1264.693,A 0.000,B 0.000,C 90.000,E1 124.692} C_DIS
LIN {X -0.051,Y -310.862,Z 1264.693,A 0.000,B 0.000,C 90.000,E1 124.659} C_DIS
LIN {X 0.060,Y -316.209,Z 1264.691,A 0.000,B 0.000,C 90.000,E1 124.405} C_DIS
LIN {X 0.141,Y -319.277,Z 1264.690,A 0.000,B 0.000,C 90.000,E1 124.119} C_DIS
LIN {X 0.052,Y -322.944,Z 1264.687,A 0.000,B 0.000,C 90.000,E1 123.627} C_DIS
LIN {X 0.132,Y -324.551,Z 1264.685,A 0.000,B 0.000,C 90.000,E1 123.293} C_DIS
LIN {X -0.040,Y -329.179,Z 1264.678,A 0.000,B 0.000,C 90.000,E1 122.054} C_DIS
LIN {X 0.163,Y -340.172,Z 1264.662,A 0.000,B 0.000,C 90.000,E1 119.205} C_DIS
LIN {X -0.101,Y -352.549,Z 1264.647,A 0.000,B 0.000,C 90.000,E1 116.488} C_DIS
LIN {X -0.014,Y -366.424,Z 1264.632,A 0.000,B 0.000,C 90.000,E1 113.770} C_DIS
LIN {X 0.064,Y -380.106,Z 1264.619,A 0.000,B 0.000,C 90.000,E1 111.408} C_DIS
LIN {X -0.160,Y -395.161,Z 1264.606,A 0.000,B 0.000,C 90.000,E1 109.141} C_DIS
LIN {X 0.106,Y -411.692,Z 1264.594,A 0.000,B 0.000,C 90.000,E1 106.858} C_DIS
LIN {X -0.244,Y -429.819,Z 1264.582,A 0.000,B 0.000,C 90.000,E1 104.717} C_DIS
LIN {X -0.115,Y -449.462,Z 1264.570,A 0.000,B 0.000,C 90.000,E1 102.591} C_DIS
LIN {X -0.213,Y -469.772,Z 1264.559,A 0.000,B 0.000,C 90.000,E1 100.658} C_DIS
LIN {X -0.213,Y -474.908,Z 1264.557,A 0.000,B 0.000,C 90.000,E1 100.197} C_DIS
LIN {X -0.169,Y -476.992,Z 1264.555,A 0.000,B 0.000,C 90.000,E1 99.962} C_DIS
LIN {X -0.125,Y -478.575,Z 1264.554,A 0.000,B 0.000,C 90.000,E1 99.726} C_DIS
LIN {X 0.141,Y -479.887,Z 1264.553,A 0.000,B 0.000,C 90.000,E1 99.443} C_DIS
LIN {X 0.013,Y -480.854,Z 1264.551,A 0.000,B 0.000,C 90.000,E1 99.208} C_DIS
LIN {X 0.172,Y -481.933,Z 1264.548,A 0.000,B 0.000,C 90.000,E1 98.690} C_DIS
LIN {X -0.069,Y -482.012,Z 1264.546,A 0.000,B 0.000,C 90.000,E1 98.219} C_DIS
LIN {X 0.104,Y -481.107,Z 1264.543,A 0.000,B 0.000,C 90.000,E1 97.701} C_DIS
LIN {X -0.199,Y -479.063,Z 1264.540,A 0.000,B 0.000,C 90.000,E1 97.239} C_DIS
LIN {X 0.151,Y -477.482,Z 1264.539,A 0.000,B 0.000,C 90.000,E1 96.947} C_DIS
LIN {X -0.048,Y -460.979,Z 1264.526,A 0.000,B 0.000,C 90.000,E1 94.702} C_DIS
LIN {X 0.185,Y -445.277,Z 1264.513,A 0.000,B 0.000,C 90.000,E1 92.350} C_DIS
LIN {X -0.149,Y -432.173,Z 1264.501,A 0.000,B 0.000,C 90.000,E1 90.286} C_DIS
LIN {X -0.004,Y -415.869,Z 1264.485,A 0.000,B 0.000,C 90.000,E1 87.306} C_DIS
LIN {X -0.104,Y -404.427,Z 1264.473,A 0.000,B 0.000,C 90.000,E1 85.122} C_DIS
LIN {X -0.100,Y -394.235,Z 1264.462,A 0.000,B 0.000,C 90.000,E1 83.166} C_DIS
LIN {X 0.170,Y -383.880,Z 1264.451,A 0.000,B 0.000,C 90.000,E1 81.141} C_DIS
LIN {X -0.109,Y -374.723,Z 1264.441,A 0.000,B 0.000,C 90.000,E1 79.454} C_DIS
LIN {X -0.099,Y -366.867,Z 1264.433,A 0.000,B 0.000,C 90.000,E1 77.993} C_DIS
LIN {X 0.184,Y -357.105,Z 1264.423,A 0.000,B 0.000,C 90.000,E1 76.172} C_DIS
LIN {X -0.046,Y -345.643,Z 1264.412,A 0.000,B 0.000,C 90.000,E1 74.102} C_DIS
LIN {X -0.014,Y -332.615,Z 1264.398,A 0.000,B 0.000,C 90.000,E1 71.638} C_DIS
LIN {X 0.167,Y -318.537,Z 1264.382,A 0.000,B 0.000,C 90.000,E1 68.773} C_DIS
LIN {X 0.108,Y -302.532,Z 1264.363,A 0.000,B 0.000,C 90.000,E1 65.229} C_DIS
LIN {X -0.074,Y -290.831,Z 1264.346,A 0.000,B 0.000,C 90.000,E1 62.281} C_DIS
LIN {X 0.015,Y -278.096,Z 1264.325,A 0.000,B 0.000,C 90.000,E1 58.535} C_DIS
LIN {X -0.112,Y -267.677,Z 1264.306,A 0.000,B 0.000,C 90.000,E1 55.102} C_DIS
LIN {X 0.063,Y -258.159,Z 1264.286,A 0.000,B 0.000,C 90.000,E1 51.537} C_DIS
LIN {X -0.033,Y -251.029,Z 1264.271,A 0.000,B 0.000,C 90.000,E1 48.690} C_DIS
LIN {X 0.001,Y -242.516,Z 1264.250,A 0.000,B 0.000,C 90.000,E1 45.040} C_DIS
LIN {X 0.006,Y -236.169,Z 1264.234,A 0.000,B 0.000,C 90.000,E1 42.081} C_DIS
LIN {X -0.026,Y -228.588,Z 1264.213,A 0.000,B 0.000,C 90.000,E1 38.338} C_DIS
LIN {X -0.041,Y -221.688,Z 1264.192,A 0.000,B 0.000,C 90.000,E1 34.532} C_DIS
LIN {X -0.042,Y -215.437,Z 1264.170,A 0.000,B 0.000,C 90.000,E1 30.669} C_DIS
LIN {X -0.003,Y -209.926,Z 1264.149,A 0.000,B 0.000,C 90.000,E1 26.744} C_DIS
LIN {X 0.051,Y -205.167,Z 1264.127,A 0.000,B 0.000,C 90.000,E1 22.770} C_DIS
LIN {X -0.068,Y -200.409,Z 1264.100,A 0.000,B 0.000,C 90.000,E1 18.000} C_DIS
LIN {X 0.035,Y -196.729,Z 1264.073,A 0.000,B 0.000,C 90.000,E1 13.119} C_DIS
LIN {X 0.050,Y -193.838,Z 1264.041,A 0.000,B 0.000,C 90.000,E1 7.409} C_DIS
LIN {X -0.045,Y -194.849,Z 1263.961,A 0.000,B 0.000,C 90.000,E1 352.989} C_DIS
LIN {X -0.052,Y -198.370,Z 1263.929,A 0.000,B 0.000,C 90.000,E1 347.285} C_DIS
LIN {X 0.003,Y -202.561,Z 1263.902,A 0.000,B 0.000,C 90.000,E1 342.417} C_DIS
LIN {X -0.004,Y -206.789,Z 1263.880,A 0.000,B 0.000,C 90.000,E1 338.411} C_DIS
LIN {X -0.073,Y -211.755,Z 1263.858,A 0.000,B 0.000,C 90.000,E1 334.460} C_DIS
LIN {X 0.011,Y -217.311,Z 1263.836,A 0.000,B 0.000,C 90.000,E1 330.511} C_DIS
LIN {X 0.028,Y -223.687,Z 1263.815,A 0.000,B 0.000,C 90.000,E1 326.628} C_DIS
LIN {X -0.140,Y -230.810,Z 1263.793,A 0.000,B 0.000,C 90.000,E1 322.844} C_DIS
LIN {X 0.111,Y -238.808,Z 1263.772,A 0.000,B 0.000,C 90.000,E1 319.013} C_DIS
LIN {X 0.041,Y -247.776,Z 1263.752,A 0.000,B 0.000,C 90.000,E1 315.324} C_DIS
LIN {X -0.122,Y -255.927,Z 1263.736,A 0.000,B 0.000,C 90.000,E1 312.447} C_DIS
LIN {X -0.083,Y -264.135,Z 1263.722,A 0.000,B 0.000,C 90.000,E1 309.930} C_DIS
LIN {X -0.069,Y -272.156,Z 1263.710,A 0.000,B 0.000,C 90.000,E1 307.810} C_DIS
LIN {X -0.173,Y -279.608,Z 1263.700,A 0.000,B 0.000,C 90.000,E1 306.091} C_DIS
LIN {X 0.158,Y -293.087,Z 1263.685,A 0.000,B 0.000,C 90.000,E1 303.293} C_DIS
LIN {X -0.102,Y -302.396,Z 1263.676,A 0.000,B 0.000,C 90.000,E1 301.671} C_DIS
LIN {X -0.041,Y -308.544,Z 1263.670,A 0.000,B 0.000,C 90.000,E1 300.669} C_DIS
LIN {X -0.065,Y -319.562,Z 1263.661,A 0.000,B 0.000,C 90.000,E1 299.077} C_DIS
LIN {X -0.080,Y -341.832,Z 1263.646,A 0.000,B 0.000,C 90.000,E1 296.232} C_DIS
LIN {X -0.206,Y -357.220,Z 1263.636,A 0.000,B 0.000,C 90.000,E1 294.463} C_DIS
LIN {X -0.005,Y -370.213,Z 1263.627,A 0.000,B 0.000,C 90.000,E1 292.950} C_DIS
LIN {X -0.203,Y -382.935,Z 1263.620,A 0.000,B 0.000,C 90.000,E1 291.535} C_DIS
LIN {X 0.003,Y -400.769,Z 1263.608,A 0.000,B 0.000,C 90.000,E1 289.504} C_DIS
LIN {X 0.102,Y -415.914,Z 1263.599,A 0.000,B 0.000,C 90.000,E1 287.873} C_DIS
LIN {X 0.004,Y -425.768,Z 1263.593,A 0.000,B 0.000,C 90.000,E1 286.804} C_DIS
LIN {X -0.234,Y -432.694,Z 1263.589,A 0.000,B 0.000,C 90.000,E1 286.024} C_DIS
LIN {X 0.013,Y -439.105,Z 1263.584,A 0.000,B 0.000,C 90.000,E1 285.190} C_DIS
LIN {X -0.114,Y -444.891,Z 1263.580,A 0.000,B 0.000,C 90.000,E1 284.411} C_DIS
LIN {X 0.137,Y -450.019,Z 1263.576,A 0.000,B 0.000,C 90.000,E1 283.592} C_DIS
LIN {X -0.004,Y -454.405,Z 1263.571,A 0.000,B 0.000,C 90.000,E1 282.827} C_DIS
LIN {X -0.103,Y -458.132,Z 1263.567,A 0.000,B 0.000,C 90.000,E1 282.063} C_DIS
LIN {X -0.176,Y -461.205,Z 1263.563,A 0.000,B 0.000,C 90.000,E1 281.299} C_DIS
LIN {X -0.152,Y -462.883,Z 1263.560,A 0.000,B 0.000,C 90.000,E1 280.782} C_DIS
LIN {X -0.027,Y -464.273,Z 1263.557,A 0.000,B 0.000,C 90.000,E1 280.254} C_DIS
LIN {X 0.104,Y -465.432,Z 1263.554,A 0.000,B 0.000,C 90.000,E1 279.726} C_DIS
LIN {X 0.167,Y -466.284,Z 1263.551,A 0.000,B 0.000,C 90.000,E1 279.208} C_DIS
LIN {X -0.222,Y -466.724,Z 1263.548,A 0.000,B 0.000,C 90.000,E1 278.746} C_DIS
LIN {X -0.076,Y -466.892,Z 1263.546,A 0.000,B 0.000,C 90.000,E1 278.219} C_DIS
LIN {X 0.005,Y -466.577,Z 1263.543,A 0.000,B 0.000,C 90.000,E1 277.701} C_DIS
LIN {X 0.088,Y -465.826,Z 1263.540,A 0.000,B 0.000,C 90.000,E1 277.182} C_DIS
LIN {X 0.171,Y -464.674,Z 1263.537,A 0.000,B 0.000,C 90.000,E1 276.663} C_DIS
LIN {X -0.213,Y -463.054,Z 1263.534,A 0.000,B 0.000,C 90.000,E1 276.201} C_DIS
LIN {X 0.140,Y -460.094,Z 1263.530,A 0.000,B 0.000,C 90.000,E1 275.391} C_DIS
LIN {X -0.037,Y -456.244,Z 1263.526,A 0.000,B 0.000,C 90.000,E1 274.645} C_DIS
LIN {X -0.045,Y -452.908,Z 1263.523,A 0.000,B 0.000,C 90.000,E1 274.131} C_DIS
LIN {X -0.035,Y -448.662,Z 1263.520,A 0.000,B 0.000,C 90.000,E1 273.612} C_DIS
LIN {X 0.167,Y -446.147,Z 1263.519,A 0.000,B 0.000,C 90.000,E1 273.326} C_DIS
LIN {X -0.051,Y -443.296,Z 1263.517,A 0.000,B 0.000,C 90.000,E1 273.094} C_DIS
LIN {X -0.193,Y -436.974,Z 1263.515,A 0.000,B 0.000,C 90.000,E1 272.636} C_DIS
LIN {X -0.185,Y -430.311,Z 1263.512,A 0.000,B 0.000,C 90.000,E1 272.236} C_DIS
LIN {X -0.118,Y -423.264,Z 1263.510,A 0.000,B 0.000,C 90.000,E1 271.892} C_DIS
LIN {X -0.018,Y -416.275,Z 1263.509,A 0.000,B 0.000,C 90.000,E1 271.604} C_DIS
LIN {X -0.018,Y -409.313,Z 1263.508,A 0.000,B 0.000,C 90.000,E1 271.375} C_DIS
LIN {X 0.033,Y -398.716,Z 1263.506,A 0.000,B 0.000,C 90.000,E1 271.088} C_DIS
LIN {X 0.182,Y -391.157,Z 1263.505,A 0.000,B 0.000,C 90.000,E1 270.917} C_DIS
LIN {X 0.125,Y -382.318,Z 1263.505,A 0.000,B 0.000,C 90.000,E1 270.802} C_DIS
LIN {X -0.118,Y -371.934,Z 1263.504,A 0.000,B 0.000,C 90.000,E1 270.745} C_DIS
LIN {X -0.003,Y -360.985,Z 1263.504,A 0.000,B 0.000,C 90.000,E1 270.688} C_DIS
LIN {X -0.035,Y -181.532,Z 1263.504,A 0.000,B 0.000,C 90.000,E1 270.688} C_DIS
LIN {X -0.079,Y -181.519,Z 1263.499,A 0.000,B 0.000,C 90.000,E1 269.828} C_DIS
LIN {X 0.084,Y -180.787,Z 1263.471,A 0.000,B 0.000,C 90.000,E1 264.723} C_DIS
LIN {X -0.022,Y -178.884,Z 1263.443,A 0.000,B 0.000,C 90.000,E1 259.690} C_DIS
LIN {X 0.054,Y -175.926,Z 1263.414,A 0.000,B 0.000,C 90.000,E1 254.574} C_DIS
LIN {X 0.000,Y -175.367,Z 1263.410,A 0.000,B 0.000,C 90.000,E1 253.740} C_DIS
LIN {X 0.058,Y -172.144,Z 1263.386,A 0.000,B 0.000,C 90.000,E1 249.444} C_DIS
LIN {X 0.035,Y -171.609,Z 1263.381,A 0.000,B 0.000,C 90.000,E1 248.592} C_DIS
LIN {X 0.024,Y -167.832,Z 1263.357,A 0.000,B 0.000,C 90.000,E1 244.280} C_DIS
LIN {X 0.041,Y -166.558,Z 1263.348,A 0.000,B 0.000,C 90.000,E1 242.538} C_DIS
LIN {X -0.049,Y -162.553,Z 1263.323,A 0.000,B 0.000,C 90.000,E1 238.201} C_DIS
LIN {X 0.011,Y -161.231,Z 1263.313,A 0.000,B 0.000,C 90.000,E1 236.421} C_DIS
LIN {X 0.046,Y -157.237,Z 1263.289,A 0.000,B 0.000,C 90.000,E1 231.984} C_DIS
LIN {X -0.031,Y -155.961,Z 1263.279,A 0.000,B 0.000,C 90.000,E1 230.231} C_DIS
LIN {X 0.027,Y -152.215,Z 1263.254,A 0.000,B 0.000,C 90.000,E1 225.729} C_DIS
LIN {X 0.048,Y -150.459,Z 1263.239,A 0.000,B 0.000,C 90.000,E1 223.014} C_DIS
LIN {X 0.073,Y -147.184,Z 1263.214,A 0.000,B 0.000,C 90.000,E1 218.463} C_DIS
LIN {X 0.040,Y -145.202,Z 1263.193,A 0.000,B 0.000,C 90.000,E1 214.818} C_DIS
LIN {X -0.050,Y -142.339,Z 1263.163,A 0.000,B 0.000,C 90.000,E1 209.333} C_DIS
LIN {X 0.004,Y -141.727,Z 1263.153,A 0.000,B 0.000,C 90.000,E1 207.462} C_DIS
LIN {X -0.014,Y -139.481,Z 1263.116,A 0.000,B 0.000,C 90.000,E1 200.972} C_DIS
LIN {X -0.025,Y -138.980,Z 1263.101,A 0.000,B 0.000,C 90.000,E1 198.181} C_DIS
LIN {X -0.040,Y -138.333,Z 1263.054,A 0.000,B 0.000,C 90.000,E1 189.782} C_DIS
LIN {X -0.040,Y -139.429,Z 1263.008,A 0.000,B 0.000,C 90.000,E1 181.375} C_DIS
LIN {X 0.013,Y -141.356,Z 1262.971,A 0.000,B 0.000,C 90.000,E1 174.837} C_DIS
LIN {X -0.011,Y -142.710,Z 1262.956,A 0.000,B 0.000,C 90.000,E1 172.064} C_DIS
LIN {X -0.052,Y -145.085,Z 1262.930,A 0.000,B 0.000,C 90.000,E1 167.465} C_DIS
LIN {X -0.056,Y -147.708,Z 1262.910,A 0.000,B 0.000,C 90.000,E1 163.795} C_DIS
LIN {X 0.028,Y -150.364,Z 1262.890,A 0.000,B 0.000,C 90.000,E1 160.115} C_DIS
LIN {X 0.046,Y -153.789,Z 1262.870,A 0.000,B 0.000,C 90.000,E1 156.485} C_DIS
LIN {X -0.035,Y -157.202,Z 1262.849,A 0.000,B 0.000,C 90.000,E1 152.922} C_DIS
LIN {X 0.048,Y -161.364,Z 1262.830,A 0.000,B 0.000,C 90.000,E1 149.331} C_DIS
LIN {X 0.059,Y -165.566,Z 1262.810,A 0.000,B 0.000,C 90.000,E1 145.801} C_DIS
LIN {X -0.057,Y -170.484,Z 1262.791,A 0.000,B 0.000,C 90.000,E1 142.351} C_DIS
LIN {X 0.091,Y -175.365,Z 1262.772,A 0.000,B 0.000,C 90.000,E1 138.852} C_DIS
LIN {X -0.045,Y -180.989,Z 1262.753,A 0.000,B 0.000,C 90.000,E1 135.486} C_DIS
LIN {X 0.080,Y -186.416,Z 1262.734,A 0.000,B 0.000,C 90.000,E1 132.081} C_DIS
LIN {X -0.120,Y -191.043,Z 1262.720,A 0.000,B 0.000,C 90.000,E1 129.644} C_DIS
LIN {X 0.072,Y -196.826,Z 1262.702,A 0.000,B 0.000,C 90.000,E1 126.297} C_DIS
LIN {X -0.022,Y -200.156,Z 1262.693,A 0.000,B 0.000,C 90.000,E1 124.659} C_DIS
LIN {X 0.169,Y -310.321,Z 1262.693,A 0.000,B 0.000,C 90.000,E1 124.612} C_DIS
LIN {X 0.065,Y -311.401,Z 1262.692,A 0.000,B 0.000,C 90.000,E1 124.612} C_DIS
LIN {X -0.083,Y -315.698,Z 1262.691,A 0.000,B 0.000,C 90.000,E1 124.452} C_DIS
LIN {X 0.028,Y -318.087,Z 1262.690,A 0.000,B 0.000,C 90.000,E1 124.246} C_DIS
LIN {X 0.075,Y -321.334,Z 1262.688,A 0.000,B 0.000,C 90.000,E1 123.865} C_DIS
LIN {X -0.054,Y -323.260,Z 1262.687,A 0.000,B 0.000,C 90.000,E1 123.579} C_DIS
LIN {X 0.087,Y -324.759,Z 1262.685,A 0.000,B 0.000,C 90.000,E1 123.245} C_DIS
LIN {X 0.003,Y -339.081,Z 1262.664,A 0.000,B 0.000,C 90.000,E1 119.489} C_DIS
LIN {X -0.127,Y -351.326,Z 1262.648,A 0.000,B 0.000,C 90.000,E1 116.744} C_DIS
LIN {X -0.076,Y -365.058,Z 1262.633,A 0.000,B 0.000,C 90.000,E1 114.027} C_DIS
LIN {X -0.030,Y -378.603,Z 1262.620,A 0.000,B 0.000,C 90.000,E1 111.663} C_DIS
LIN {X 0.083,Y -393.511,Z 1262.608,A 0.000,B 0.000,C 90.000,E1 109.341} C_DIS
LIN {X 0.061,Y -409.885,Z 1262.595,A 0.000,B 0.000,C 90.000,E1 107.094} C_DIS
LIN {X 0.076,Y -427.840,Z 1262.583,A 0.000,B 0.000,C 90.000,E1 104.898} C_DIS
LIN {X 0.127,Y -447.360,Z 1262.571,A 0.000,B 0.000,C 90.000,E1 102.771} C_DIS
LIN {X -0.097,Y -467.614,Z 1262.560,A 0.000,B 0.000,C 90.000,E1 100.838} C_DIS
LIN {X -0.059,Y -475.252,Z 1262.556,A 0.000,B 0.000,C 90.000,E1 100.141} C_DIS
LIN {X 0.008,Y -477.196,Z 1262.555,A 0.000,B 0.000,C 90.000,E1 99.905} C_DIS
LIN {X -0.124,Y -478.822,Z 1262.554,A 0.000,B 0.000,C 90.000,E1 99.670} C_DIS
LIN {X 0.215,Y -480.039,Z 1262.552,A 0.000,B 0.000,C 90.000,E1 99.378} C_DIS
LIN {X -0.109,Y -481.525,Z 1262.549,A 0.000,B 0.000,C 90.000,E1 98.916} C_DIS
LIN {X 0.051,Y -481.964,Z 1262.547,A 0.000,B 0.000,C 90.000,E1 98.398} C_DIS
LIN {X -0.255,Y -481.430,Z 1262.544,A 0.000,B 0.000,C 90.000,E1 97.936} C_DIS
LIN {X -0.018,Y -479.839,Z 1262.541,A 0.000,B 0.000,C 90.000,E1 97.409} C_DIS
LIN {X -0.201,Y -478.561,Z 1262.540,A 0.000,B 0.000,C 90.000,E1 97.182} C_DIS
LIN {X -0.038,Y -474.921,Z 1262.537,A 0.000,B 0.000,C 90.000,E1 96.663} C_DIS
LIN {X 0.215,Y -455.098,Z 1262.521,A 0.000,B 0.000,C 90.000,E1 93.841} C_DIS
LIN {X -0.073,Y -434.749,Z 1262.504,A 0.000,B 0.000,C 90.000,E1 90.745} C_DIS
LIN {X -0.065,Y -415.339,Z 1262.485,A 0.000,B 0.000,C 90.000,E1 87.249} C_DIS
LIN {X -0.177,Y -403.898,Z 1262.472,A 0.000,B 0.000,C 90.000,E1 85.065} C_DIS
LIN {X -0.178,Y -393.687,Z 1262.462,A 0.000,B 0.000,C 90.000,E1 83.109} C_DIS
LIN {X 0.076,Y -383.350,Z 1262.451,A 0.000,B 0.000,C 90.000,E1 81.084} C_DIS
LIN {X 0.156,Y -374.174,Z 1262.441,A 0.000,B 0.000,C 90.000,E1 79.342} C_DIS
LIN {X 0.153,Y -366.310,Z 1262.433,A 0.000,B 0.000,C 90.000,E1 77.881} C_DIS
LIN {X 0.068,Y -356.573,Z 1262.423,A 0.000,B 0.000,C 90.000,E1 76.117} C_DIS
LIN {X -0.084,Y -345.113,Z 1262.411,A 0.000,B 0.000,C 90.000,E1 74.031} C_DIS
LIN {X -0.157,Y -332.094,Z 1262.398,A 0.000,B 0.000,C 90.000,E1 71.583} C_DIS
LIN {X -0.047,Y -316.540,Z 1262.380,A 0.000,B 0.000,C 90.000,E1 68.411} C_DIS
LIN {X -0.062,Y -302.117,Z 1262.362,A 0.000,B 0.000,C 90.000,E1 65.177} C_DIS
LIN {X 0.140,Y -290.448,Z 1262.345,A 0.000,B 0.000,C 90.000,E1 62.153} C_DIS
LIN {X 0.007,Y -278.800,Z 1262.327,A 0.000,B 0.000,C 90.000,E1 58.791} C_DIS
LIN {X -0.023,Y -268.247,Z 1262.307,A 0.000,B 0.000,C 90.000,E1 55.341} C_DIS
LIN {X -0.046,Y -258.619,Z 1262.288,A 0.000,B 0.000,C 90.000,E1 51.823} C_DIS
LIN {X -0.079,Y -249.700,Z 1262.268,A 0.000,B 0.000,C 90.000,E1 48.243} C_DIS
LIN {X -0.091,Y -241.257,Z 1262.248,A 0.000,B 0.000,C 90.000,E1 44.595} C_DIS
LIN {X 0.049,Y -234.945,Z 1262.231,A 0.000,B 0.000,C 90.000,E1 41.595} C_DIS
LIN {X -0.033,Y -227.395,Z 1262.210,A 0.000,B 0.000,C 90.000,E1 37.855} C_DIS
LIN {X -0.046,Y -220.509,Z 1262.189,A 0.000,B 0.000,C 90.000,E1 34.040} C_DIS
LIN {X 0.096,Y -214.301,Z 1262.167,A 0.000,B 0.000,C 90.000,E1 30.129} C_DIS
LIN {X -0.004,Y -208.870,Z 1262.146,A 0.000,B 0.000,C 90.000,E1 26.232} C_DIS
LIN {X -0.065,Y -204.189,Z 1262.124,A 0.000,B 0.000,C 90.000,E1 22.280} C_DIS
LIN {X -0.027,Y -199.531,Z 1262.097,A 0.000,B 0.000,C 90.000,E1 17.457} C_DIS
LIN {X -0.008,Y -195.979,Z 1262.070,A 0.000,B 0.000,C 90.000,E1 12.591} C_DIS
LIN {X -0.054,Y -193.298,Z 1262.038,A 0.000,B 0.000,C 90.000,E1 6.891} C_DIS
LIN {X -0.030,Y -194.272,Z 1261.965,A 0.000,B 0.000,C 90.000,E1 353.799} C_DIS
LIN {X 0.094,Y -197.589,Z 1261.934,A 0.000,B 0.000,C 90.000,E1 348.049} C_DIS
LIN {X 0.069,Y -201.660,Z 1261.907,A 0.000,B 0.000,C 90.000,E1 343.196} C_DIS
LIN {X -0.036,Y -206.670,Z 1261.880,A 0.000,B 0.000,C 90.000,E1 338.411} C_DIS
LIN {X 0.082,Y -211.665,Z 1261.858,A 0.000,B 0.000,C 90.000,E1 334.409} C_DIS
LIN {X -0.029,Y -217.249,Z 1261.836,A 0.000,B 0.000,C 90.000,E1 330.511} C_DIS
LIN {X -0.015,Y -223.648,Z 1261.815,A 0.000,B 0.000,C 90.000,E1 326.628} C_DIS
LIN {X -0.002,Y -230.785,Z 1261.793,A 0.000,B 0.000,C 90.000,E1 322.798} C_DIS
LIN {X 0.063,Y -238.771,Z 1261.772,A 0.000,B 0.000,C 90.000,E1 319.013} C_DIS
LIN {X -0.010,Y -247.727,Z 1261.752,A 0.000,B 0.000,C 90.000,E1 315.324} C_DIS
LIN {X 0.013,Y -255.874,Z 1261.736,A 0.000,B 0.000,C 90.000,E1 312.405} C_DIS
LIN {X -0.087,Y -265.342,Z 1261.720,A 0.000,B 0.000,C 90.000,E1 309.564} C_DIS
LIN {X -0.050,Y -273.535,Z 1261.708,A 0.000,B 0.000,C 90.000,E1 307.443} C_DIS
LIN {X -0.128,Y -281.170,Z 1261.698,A 0.000,B 0.000,C 90.000,E1 305.724} C_DIS
LIN {X 0.093,Y -293.021,Z 1261.685,A 0.000,B 0.000,C 90.000,E1 303.293} C_DIS
LIN {X -0.171,Y -302.327,Z 1261.676,A 0.000,B 0.000,C 90.000,E1 301.671} C_DIS
LIN {X -0.112,Y -308.462,Z 1261.670,A 0.000,B 0.000,C 90.000,E1 300.669} C_DIS
LIN {X -0.007,Y -319.295,Z 1261.661,A 0.000,B 0.000,C 90.000,E1 299.077} C_DIS
LIN {X -0.028,Y -341.549,Z 1261.646,A 0.000,B 0.000,C 90.000,E1 296.232} C_DIS
LIN {X 0.051,Y -357.346,Z 1261.635,A 0.000,B 0.000,C 90.000,E1 294.387} C_DIS
LIN {X 0.156,Y -370.289,Z 1261.627,A 0.000,B 0.000,C 90.000,E1 292.898} C_DIS
LIN {X 0.103,Y -382.871,Z 1261.619,A 0.000,B 0.000,C 90.000,E1 291.482} C_DIS
LIN {X 0.016,Y -400.685,Z 1261.608,A 0.000,B 0.000,C 90.000,E1 289.504} C_DIS
LIN {X -0.022,Y -416.049,Z 1261.599,A 0.000,B 0.000,C 90.000,E1 287.873} C_DIS
LIN {X -0.140,Y -425.915,Z 1261.593,A 0.000,B 0.000,C 90.000,E1 286.804} C_DIS
LIN {X 0.037,Y -432.815,Z 1261.589,A 0.000,B 0.000,C 90.000,E1 285.969} C_DIS
LIN {X -0.133,Y -439.210,Z 1261.584,A 0.000,B 0.000,C 90.000,E1 285.190} C_DIS
LIN {X 0.170,Y -444.969,Z 1261.580,A 0.000,B 0.000,C 90.000,E1 284.356} C_DIS
LIN {X -0.011,Y -450.056,Z 1261.576,A 0.000,B 0.000,C 90.000,E1 283.592} C_DIS
LIN {X -0.153,Y -454.449,Z 1261.571,A 0.000,B 0.000,C 90.000,E1 282.827} C_DIS
LIN {X 0.196,Y -458.176,Z 1261.567,A 0.000,B 0.000,C 90.000,E1 282.007} C_DIS
LIN {X 0.126,Y -461.224,Z 1261.563,A 0.000,B 0.000,C 90.000,E1 281.243} C_DIS
LIN {X 0.153,Y -462.900,Z 1261.560,A 0.000,B 0.000,C 90.000,E1 280.725} C_DIS
LIN {X -0.178,Y -464.291,Z 1261.557,A 0.000,B 0.000,C 90.000,E1 280.254} C_DIS
LIN {X -0.047,Y -465.431,Z 1261.554,A 0.000,B 0.000,C 90.000,E1 279.726} C_DIS
LIN {X 0.016,Y -466.297,Z 1261.551,A 0.000,B 0.000,C 90.000,E1 279.208} C_DIS
LIN {X 0.089,Y -466.803,Z 1261.548,A 0.000,B 0.000,C 90.000,E1 278.690} C_DIS
LIN {X 0.235,Y -466.949,Z 1261.546,A 0.000,B 0.000,C 90.000,E1 278.163} C_DIS
LIN {X -0.145,Y -466.644,Z 1261.543,A 0.000,B 0.000,C 90.000,E1 277.701} C_DIS
LIN {X -0.062,Y -465.947,Z 1261.540,A 0.000,B 0.000,C 90.000,E1 277.182} C_DIS
LIN {X 0.021,Y -464.785,Z 1261.537,A 0.000,B 0.000,C 90.000,E1 276.663} C_DIS
LIN {X 0.100,Y -463.192,Z 1261.534,A 0.000,B 0.000,C 90.000,E1 276.144} C_DIS
LIN {X -0.005,Y -460.231,Z 1261.530,A 0.000,B 0.000,C 90.000,E1 275.391} C_DIS
LIN {X 0.006,Y -457.818,Z 1261.527,A 0.000,B 0.000,C 90.000,E1 274.878} C_DIS
LIN {X 0.042,Y -454.800,Z 1261.524,A 0.000,B 0.000,C 90.000,E1 274.359} C_DIS
LIN {X 0.059,Y -451.092,Z 1261.521,A 0.000,B 0.000,C 90.000,E1 273.841} C_DIS
LIN {X 0.029,Y -446.311,Z 1261.519,A 0.000,B 0.000,C 90.000,E1 273.326} C_DIS
LIN {X -0.188,Y -443.493,Z 1261.517,A 0.000,B 0.000,C 90.000,E1 273.094} C_DIS
LIN {X 0.082,Y -437.133,Z 1261.514,A 0.000,B 0.000,C 90.000,E1 272.579} C_DIS
LIN {X 0.070,Y -430.435,Z 1261.512,A 0.000,B 0.000,C 90.000,E1 272.178} C_DIS
LIN {X 0.140,Y -423.408,Z 1261.510,A 0.000,B 0.000,C 90.000,E1 271.835} C_DIS
LIN {X -0.195,Y -416.368,Z 1261.509,A 0.000,B 0.000,C 90.000,E1 271.604} C_DIS
LIN {X -0.072,Y -406.073,Z 1261.507,A 0.000,B 0.000,C 90.000,E1 271.260} C_DIS
LIN {X -0.120,Y -398.828,Z 1261.506,A 0.000,B 0.000,C 90.000,E1 271.088} C_DIS
LIN {X 0.031,Y -391.281,Z 1261.505,A 0.000,B 0.000,C 90.000,E1 270.917} C_DIS
LIN {X -0.023,Y -382.507,Z 1261.504,A 0.000,B 0.000,C 90.000,E1 270.802} C_DIS
LIN {X -0.017,Y -368.787,Z 1261.504,A 0.000,B 0.000,C 90.000,E1 270.688} C_DIS
LIN {X -0.141,Y -361.577,Z 1261.504,A 0.000,B 0.000,C 90.000,E1 270.688} C_DIS
LIN {X 0.079,Y -181.537,Z 1261.504,A 0.000,B 0.000,C 90.000,E1 270.630} C_DIS
LIN {X 0.039,Y -181.513,Z 1261.499,A 0.000,B 0.000,C 90.000,E1 269.771} C_DIS
LIN {X 0.022,Y -180.779,Z 1261.471,A 0.000,B 0.000,C 90.000,E1 264.723} C_DIS
LIN {X -0.083,Y -178.875,Z 1261.443,A 0.000,B 0.000,C 90.000,E1 259.690} C_DIS
LIN {X -0.007,Y -175.918,Z 1261.414,A 0.000,B 0.000,C 90.000,E1 254.574} C_DIS
LIN {X 0.048,Y -174.613,Z 1261.405,A 0.000,B 0.000,C 90.000,E1 252.851} C_DIS
LIN {X -0.025,Y -171.594,Z 1261.381,A 0.000,B 0.000,C 90.000,E1 248.592} C_DIS
LIN {X -0.036,Y -167.816,Z 1261.357,A 0.000,B 0.000,C 90.000,E1 244.280} C_DIS
LIN {X -0.018,Y -166.539,Z 1261.347,A 0.000,B 0.000,C 90.000,E1 242.538} C_DIS
LIN {X 0.031,Y -162.536,Z 1261.323,A 0.000,B 0.000,C 90.000,E1 238.152} C_DIS
LIN {X -0.047,Y -161.212,Z 1261.313,A 0.000,B 0.000,C 90.000,E1 236.421} C_DIS
LIN {X -0.012,Y -157.221,Z 1261.289,A 0.000,B 0.000,C 90.000,E1 231.984} C_DIS
LIN {X 0.011,Y -155.947,Z 1261.279,A 0.000,B 0.000,C 90.000,E1 230.194} C_DIS
LIN {X -0.030,Y -152.200,Z 1261.254,A 0.000,B 0.000,C 90.000,E1 225.729} C_DIS
LIN {X -0.008,Y -150.445,Z 1261.239,A 0.000,B 0.000,C 90.000,E1 223.014} C_DIS
LIN {X 0.018,Y -147.171,Z 1261.214,A 0.000,B 0.000,C 90.000,E1 218.463} C_DIS
LIN {X -0.014,Y -145.187,Z 1261.193,A 0.000,B 0.000,C 90.000,E1 214.818} C_DIS
LIN {X 0.021,Y -142.331,Z 1261.163,A 0.000,B 0.000,C 90.000,E1 209.283} C_DIS
LIN {X -0.051,Y -141.719,Z 1261.152,A 0.000,B 0.000,C 90.000,E1 207.462} C_DIS
LIN {X 0.062,Y -139.476,Z 1261.116,A 0.000,B 0.000,C 90.000,E1 200.918} C_DIS
LIN {X 0.053,Y -138.973,Z 1261.101,A 0.000,B 0.000,C 90.000,E1 198.127} C_DIS
LIN {X 0.043,Y -138.330,Z 1261.054,A 0.000,B 0.000,C 90.000,E1 189.726} C_DIS
LIN {X 0.046,Y -139.434,Z 1261.007,A 0.000,B 0.000,C 90.000,E1 181.318} C_DIS
LIN {X -0.014,Y -140.962,Z 1260.976,A 0.000,B 0.000,C 90.000,E1 175.755} C_DIS
LIN {X 0.077,Y -142.719,Z 1260.956,A 0.000,B 0.000,C 90.000,E1 172.008} C_DIS
LIN {X 0.036,Y -145.098,Z 1260.930,A 0.000,B 0.000,C 90.000,E1 167.409} C_DIS
LIN {X 0.030,Y -147.722,Z 1260.910,A 0.000,B 0.000,C 90.000,E1 163.740} C_DIS
LIN {X -0.029,Y -150.381,Z 1260.890,A 0.000,B 0.000,C 90.000,E1 160.115} C_DIS
LIN {X -0.012,Y -153.812,Z 1260.869,A 0.000,B 0.000,C 90.000,E1 156.485} C_DIS
LIN {X 0.048,Y -157.223,Z 1260.849,A 0.000,B 0.000,C 90.000,E1 152.871} C_DIS
LIN {X -0.011,Y -161.390,Z 1260.830,A 0.000,B 0.000,C 90.000,E1 149.331} C_DIS
LIN {X -0.001,Y -165.592,Z 1260.810,A 0.000,B 0.000,C 90.000,E1 145.801} C_DIS
LIN {X -0.014,Y -170.515,Z 1260.791,A 0.000,B 0.000,C 90.000,E1 142.316} C_DIS
LIN {X 0.030,Y -175.395,Z 1260.771,A 0.000,B 0.000,C 90.000,E1 138.852} C_DIS
LIN {X 0.021,Y -181.019,Z 1260.753,A 0.000,B 0.000,C 90.000,E1 135.445} C_DIS
LIN {X 0.015,Y -186.450,Z 1260.734,A 0.000,B 0.000,C 90.000,E1 132.081} C_DIS
LIN {X 0.085,Y -191.074,Z 1260.720,A 0.000,B 0.000,C 90.000,E1 129.564} C_DIS
LIN {X 0.006,Y -196.863,Z 1260.702,A 0.000,B 0.000,C 90.000,E1 126.297} C_DIS
LIN {X 0.111,Y -200.176,Z 1260.693,A 0.000,B 0.000,C 90.000,E1 124.612} C_DIS
LIN {X 0.119,Y -309.499,Z 1260.692,A 0.000,B 0.000,C 90.000,E1 124.612} C_DIS
LIN {X -0.039,Y -311.517,Z 1260.692,A 0.000,B 0.000,C 90.000,E1 124.612} C_DIS
LIN {X 0.072,Y -315.763,Z 1260.691,A 0.000,B 0.000,C 90.000,E1 124.405} C_DIS
LIN {X -0.078,Y -318.143,Z 1260.690,A 0.000,B 0.000,C 90.000,E1 124.246} C_DIS
LIN {X -0.031,Y -321.383,Z 1260.688,A 0.000,B 0.000,C 90.000,E1 123.865} C_DIS
LIN {X -0.163,Y -323.310,Z 1260.686,A 0.000,B 0.000,C 90.000,E1 123.579} C_DIS
LIN {X -0.026,Y -324.809,Z 1260.685,A 0.000,B 0.000,C 90.000,E1 123.245} C_DIS
LIN {X 0.055,Y -339.140,Z 1260.664,A 0.000,B 0.000,C 90.000,E1 119.461} C_DIS
LIN {X 0.069,Y -351.394,Z 1260.648,A 0.000,B 0.000,C 90.000,E1 116.693} C_DIS
LIN {X -0.048,Y -365.136,Z 1260.633,A 0.000,B 0.000,C 90.000,E1 114.003} C_DIS
LIN {X -0.013,Y -378.692,Z 1260.620,A 0.000,B 0.000,C 90.000,E1 111.642} C_DIS
LIN {X 0.088,Y -393.611,Z 1260.607,A 0.000,B 0.000,C 90.000,E1 109.322} C_DIS
LIN {X -0.067,Y -409.996,Z 1260.595,A 0.000,B 0.000,C 90.000,E1 107.094} C_DIS
LIN {X -0.054,Y -427.964,Z 1260.583,A 0.000,B 0.000,C 90.000,E1 104.898} C_DIS
LIN {X -0.003,Y -447.494,Z 1260.571,A 0.000,B 0.000,C 90.000,E1 102.771} C_DIS
LIN {X -0.222,Y -467.753,Z 1260.560,A 0.000,B 0.000,C 90.000,E1 100.838} C_DIS
LIN {X -0.184,Y -475.352,Z 1260.556,A 0.000,B 0.000,C 90.000,E1 100.141} C_DIS
LIN {X -0.116,Y -477.241,Z 1260.555,A 0.000,B 0.000,C 90.000,E1 99.905} C_DIS
LIN {X 0.224,Y -478.823,Z 1260.554,A 0.000,B 0.000,C 90.000,E1 99.613} C_DIS
LIN {X 0.092,Y -480.008,Z 1260.552,A 0.000,B 0.000,C 90.000,E1 99.378} C_DIS
LIN {X -0.233,Y -481.442,Z 1260.549,A 0.000,B 0.000,C 90.000,E1 98.916} C_DIS
LIN {X -0.073,Y -481.836,Z 1260.547,A 0.000,B 0.000,C 90.000,E1 98.398} C_DIS
LIN {X 0.163,Y -481.256,Z 1260.544,A 0.000,B 0.000,C 90.000,E1 97.871} C_DIS
LIN {X -0.142,Y -479.612,Z 1260.541,A 0.000,B 0.000,C 90.000,E1 97.409} C_DIS
LIN {X 0.149,Y -478.300,Z 1260.540,A 0.000,B 0.000,C 90.000,E1 97.125} C_DIS
LIN {X 0.175,Y -472.732,Z 1260.536,A 0.000,B 0.000,C 90.000,E1 96.372} C_DIS
LIN {X 0.087,Y -454.791,Z 1260.521,A 0.000,B 0.000,C 90.000,E1 93.841} C_DIS
LIN {X -0.207,Y -434.460,Z 1260.504,A 0.000,B 0.000,C 90.000,E1 90.745} C_DIS
LIN {X -0.203,Y -415.062,Z 1260.485,A 0.000,B 0.000,C 90.000,E1 87.249} C_DIS
LIN {X 0.085,Y -403.614,Z 1260.472,A 0.000,B 0.000,C 90.000,E1 85.008} C_DIS
LIN {X 0.068,Y -393.413,Z 1260.461,A 0.000,B 0.000,C 90.000,E1 83.053} C_DIS
LIN {X -0.070,Y -383.071,Z 1260.450,A 0.000,B 0.000,C 90.000,E1 81.084} C_DIS
LIN {X 0.010,Y -373.909,Z 1260.441,A 0.000,B 0.000,C 90.000,E1 79.342} C_DIS
LIN {X -0.013,Y -364.421,Z 1260.431,A 0.000,B 0.000,C 90.000,E1 77.589} C_DIS
LIN {X -0.042,Y -354.694,Z 1260.421,A 0.000,B 0.000,C 90.000,E1 75.811} C_DIS
LIN {X 0.019,Y -343.235,Z 1260.409,A 0.000,B 0.000,C 90.000,E1 73.685} C_DIS
LIN {X -0.038,Y -328.657,Z 1260.394,A 0.000,B 0.000,C 90.000,E1 70.913} C_DIS
LIN {X 0.083,Y -313.321,Z 1260.376,A 0.000,B 0.000,C 90.000,E1 67.720} C_DIS
LIN {X 0.097,Y -299.224,Z 1260.358,A 0.000,B 0.000,C 90.000,E1 64.460} C_DIS
LIN {X -0.167,Y -287.834,Z 1260.342,A 0.000,B 0.000,C 90.000,E1 61.513} C_DIS
LIN {X 0.006,Y -276.393,Z 1260.323,A 0.000,B 0.000,C 90.000,E1 58.074} C_DIS
LIN {X -0.026,Y -265.979,Z 1260.303,A 0.000,B 0.000,C 90.000,E1 54.609} C_DIS
LIN {X -0.111,Y -256.490,Z 1260.284,A 0.000,B 0.000,C 90.000,E1 51.090} C_DIS
LIN {X -0.045,Y -247.661,Z 1260.264,A 0.000,B 0.000,C 90.000,E1 47.472} C_DIS
LIN {X 0.044,Y -239.348,Z 1260.243,A 0.000,B 0.000,C 90.000,E1 43.785} C_DIS
LIN {X -0.029,Y -233.037,Z 1260.227,A 0.000,B 0.000,C 90.000,E1 40.825} C_DIS
LIN {X 0.047,Y -225.592,Z 1260.206,A 0.000,B 0.000,C 90.000,E1 37.030} C_DIS
LIN {X -0.017,Y -218.793,Z 1260.184,A 0.000,B 0.000,C 90.000,E1 33.214} C_DIS
LIN {X -0.041,Y -212.663,Z 1260.163,A 0.000,B 0.000,C 90.000,E1 29.333} C_DIS
LIN {X -0.097,Y -207.390,Z 1260.141,A 0.000,B 0.000,C 90.000,E1 25.412} C_DIS
LIN {X -0.014,Y -202.883,Z 1260.119,A 0.000,B 0.000,C 90.000,E1 21.408} C_DIS
LIN {X 0.033,Y -198.416,Z 1260.092,A 0.000,B 0.000,C 90.000,E1 16.567} C_DIS
LIN {X -0.014,Y -194.581,Z 1260.061,A 0.000,B 0.000,C 90.000,E1 10.894} C_DIS
LIN {X 0.070,Y -192.287,Z 1260.020,A 0.000,B 0.000,C 90.000,E1 3.498} C_DIS
LIN {X -0.041,Y -194.056,Z 1259.965,A 0.000,B 0.000,C 90.000,E1 353.799} C_DIS
LIN {X 0.074,Y -197.422,Z 1259.934,A 0.000,B 0.000,C 90.000,E1 348.049} C_DIS
LIN {X 0.042,Y -201.504,Z 1259.907,A 0.000,B 0.000,C 90.000,E1 343.196} C_DIS
LIN {X -0.070,Y -206.550,Z 1259.880,A 0.000,B 0.000,C 90.000,E1 338.411} C_DIS
LIN {X 0.044,Y -211.574,Z 1259.858,A 0.000,B 0.000,C 90.000,E1 334.409} C_DIS
LIN {X 0.119,Y -217.188,Z 1259.836,A 0.000,B 0.000,C 90.000,E1 330.461} C_DIS
LIN {X -0.059,Y -223.593,Z 1259.815,A 0.000,B 0.000,C 90.000,E1 326.628} C_DIS
LIN {X 0.090,Y -230.745,Z 1259.793,A 0.000,B 0.000,C 90.000,E1 322.763} C_DIS
LIN {X 0.012,Y -238.731,Z 1259.772,A 0.000,B 0.000,C 90.000,E1 319.013} C_DIS
LIN {X -0.064,Y -247.687,Z 1259.752,A 0.000,B 0.000,C 90.000,E1 315.324} C_DIS
LIN {X 0.129,Y -255.822,Z 1259.735,A 0.000,B 0.000,C 90.000,E1 312.366} C_DIS
LIN {X 0.004,Y -264.041,Z 1259.722,A 0.000,B 0.000,C 90.000,E1 309.886} C_DIS
LIN {X 0.112,Y -270.646,Z 1259.712,A 0.000,B 0.000,C 90.000,E1 308.096} C_DIS
LIN {X -0.007,Y -277.951,Z 1259.702,A 0.000,B 0.000,C 90.000,E1 306.377} C_DIS
LIN {X -0.091,Y -289.445,Z 1259.689,A 0.000,B 0.000,C 90.000,E1 303.992} C_DIS
LIN {X 0.000,Y -300.300,Z 1259.677,A 0.000,B 0.000,C 90.000,E1 301.957} C_DIS
LIN {X -0.187,Y -308.381,Z 1259.670,A 0.000,B 0.000,C 90.000,E1 300.669} C_DIS
LIN {X -0.150,Y -319.290,Z 1259.661,A 0.000,B 0.000,C 90.000,E1 299.077} C_DIS
LIN {X -0.180,Y -341.542,Z 1259.646,A 0.000,B 0.000,C 90.000,E1 296.232} C_DIS
LIN {X -0.058,Y -357.288,Z 1259.635,A 0.000,B 0.000,C 90.000,E1 294.387} C_DIS
LIN {X 0.014,Y -370.316,Z 1259.627,A 0.000,B 0.000,C 90.000,E1 292.898} C_DIS
LIN {X -0.005,Y -383.066,Z 1259.619,A 0.000,B 0.000,C 90.000,E1 291.461} C_DIS
LIN {X 0.125,Y -400.963,Z 1259.608,A 0.000,B 0.000,C 90.000,E1 289.450} C_DIS
LIN {X 0.063,Y -416.416,Z 1259.599,A 0.000,B 0.000,C 90.000,E1 287.819} C_DIS
LIN {X 0.077,Y -426.263,Z 1259.593,A 0.000,B 0.000,C 90.000,E1 286.732} C_DIS
LIN {X 0.257,Y -433.127,Z 1259.589,A 0.000,B 0.000,C 90.000,E1 285.898} C_DIS
LIN {X -0.026,Y -439.477,Z 1259.584,A 0.000,B 0.000,C 90.000,E1 285.134} C_DIS
LIN {X -0.150,Y -445.196,Z 1259.580,A 0.000,B 0.000,C 90.000,E1 284.356} C_DIS
LIN {X 0.106,Y -450.251,Z 1259.575,A 0.000,B 0.000,C 90.000,E1 283.536} C_DIS
LIN {X -0.031,Y -454.606,Z 1259.571,A 0.000,B 0.000,C 90.000,E1 282.771} C_DIS
LIN {X -0.127,Y -458.261,Z 1259.567,A 0.000,B 0.000,C 90.000,E1 282.007} C_DIS
LIN {X -0.198,Y -461.317,Z 1259.562,A 0.000,B 0.000,C 90.000,E1 281.243} C_DIS
LIN {X -0.086,Y -462.980,Z 1259.559,A 0.000,B 0.000,C 90.000,E1 280.715} C_DIS
LIN {X -0.046,Y -464.379,Z 1259.557,A 0.000,B 0.000,C 90.000,E1 280.197} C_DIS
LIN {X 0.087,Y -465.510,Z 1259.554,A 0.000,B 0.000,C 90.000,E1 279.670} C_DIS
LIN {X 0.150,Y -466.375,Z 1259.551,A 0.000,B 0.000,C 90.000,E1 279.151} C_DIS
LIN {X -0.167,Y -466.859,Z 1259.548,A 0.000,B 0.000,C 90.000,E1 278.681} C_DIS
LIN {X -0.089,Y -466.974,Z 1259.545,A 0.000,B 0.000,C 90.000,E1 278.163} C_DIS
LIN {X -0.008,Y -466.710,Z 1259.542,A 0.000,B 0.000,C 90.000,E1 277.644} C_DIS
LIN {X 0.076,Y -465.993,Z 1259.540,A 0.000,B 0.000,C 90.000,E1 277.125} C_DIS
LIN {X 0.160,Y -464.816,Z 1259.537,A 0.000,B 0.000,C 90.000,E1 276.606} C_DIS
LIN {X -0.221,Y -463.263,Z 1259.534,A 0.000,B 0.000,C 90.000,E1 276.144} C_DIS
LIN {X -0.148,Y -461.388,Z 1259.531,A 0.000,B 0.000,C 90.000,E1 275.625} C_DIS
LIN {X 0.145,Y -457.870,Z 1259.527,A 0.000,B 0.000,C 90.000,E1 274.821} C_DIS
LIN {X 0.181,Y -454.815,Z 1259.524,A 0.000,B 0.000,C 90.000,E1 274.302} C_DIS
LIN {X 0.198,Y -451.086,Z 1259.521,A 0.000,B 0.000,C 90.000,E1 273.784} C_DIS
LIN {X 0.166,Y -446.273,Z 1259.518,A 0.000,B 0.000,C 90.000,E1 273.269} C_DIS
LIN {X -0.052,Y -443.396,Z 1259.517,A 0.000,B 0.000,C 90.000,E1 273.037} C_DIS
LIN {X -0.112,Y -440.432,Z 1259.516,A 0.000,B 0.000,C 90.000,E1 272.808} C_DIS
LIN {X 0.067,Y -433.936,Z 1259.513,A 0.000,B 0.000,C 90.000,E1 272.350} C_DIS
LIN {X -0.078,Y -427.116,Z 1259.511,A 0.000,B 0.000,C 90.000,E1 272.007} C_DIS
LIN {X -0.199,Y -420.119,Z 1259.509,A 0.000,B 0.000,C 90.000,E1 271.718} C_DIS
LIN {X 0.025,Y -412.954,Z 1259.508,A 0.000,B 0.000,C 90.000,E1 271.432} C_DIS
LIN {X 0.129,Y -405.990,Z 1259.507,A 0.000,B 0.000,C 90.000,E1 271.203} C_DIS
LIN {X 0.079,Y -398.622,Z 1259.506,A 0.000,B 0.000,C 90.000,E1 271.031} C_DIS
LIN {X -0.137,Y -391.238,Z 1259.505,A 0.000,B 0.000,C 90.000,E1 270.917} C_DIS
LIN {X -0.170,Y -382.663,Z 1259.504,A 0.000,B 0.000,C 90.000,E1 270.802} C_DIS
LIN {X -0.157,Y -368.825,Z 1259.504,A 0.000,B 0.000,C 90.000,E1 270.688} C_DIS
LIN {X 0.083,Y -361.478,Z 1259.504,A 0.000,B 0.000,C 90.000,E1 270.630} C_DIS
LIN {X 0.010,Y -181.542,Z 1259.504,A 0.000,B 0.000,C 90.000,E1 270.630} C_DIS
LIN {X -0.030,Y -181.508,Z 1259.499,A 0.000,B 0.000,C 90.000,E1 269.771} C_DIS
LIN {X 0.075,Y -180.907,Z 1259.475,A 0.000,B 0.000,C 90.000,E1 265.527} C_DIS
LIN {X -0.047,Y -180.771,Z 1259.471,A 0.000,B 0.000,C 90.000,E1 264.723} C_DIS
LIN {X 0.024,Y -178.865,Z 1259.443,A 0.000,B 0.000,C 90.000,E1 259.634} C_DIS
LIN {X -0.075,Y -175.908,Z 1259.414,A 0.000,B 0.000,C 90.000,E1 254.574} C_DIS
LIN {X -0.018,Y -174.595,Z 1259.405,A 0.000,B 0.000,C 90.000,E1 252.851} C_DIS
LIN {X 0.067,Y -171.577,Z 1259.381,A 0.000,B 0.000,C 90.000,E1 248.539} C_DIS
LIN {X 0.049,Y -167.799,Z 1259.357,A 0.000,B 0.000,C 90.000,E1 244.229} C_DIS
LIN {X 0.063,Y -166.518,Z 1259.347,A 0.000,B 0.000,C 90.000,E1 242.487} C_DIS
LIN {X 0.051,Y -162.519,Z 1259.323,A 0.000,B 0.000,C 90.000,E1 238.122} C_DIS
LIN {X 0.023,Y -161.191,Z 1259.313,A 0.000,B 0.000,C 90.000,E1 236.373} C_DIS
LIN {X -0.074,Y -157.203,Z 1259.289,A 0.000,B 0.000,C 90.000,E1 231.984} C_DIS
LIN {X -0.052,Y -155.930,Z 1259.279,A 0.000,B 0.000,C 90.000,E1 230.194} C_DIS
LIN {X -0.092,Y -152.182,Z 1259.254,A 0.000,B 0.000,C 90.000,E1 225.729} C_DIS
LIN {X 0.032,Y -150.429,Z 1259.239,A 0.000,B 0.000,C 90.000,E1 222.975} C_DIS
LIN {X -0.042,Y -147.157,Z 1259.214,A 0.000,B 0.000,C 90.000,E1 218.463} C_DIS
LIN {X -0.075,Y -145.172,Z 1259.193,A 0.000,B 0.000,C 90.000,E1 214.818} C_DIS
LIN {X -0.038,Y -142.322,Z 1259.163,A 0.000,B 0.000,C 90.000,E1 209.283} C_DIS
LIN {X 0.082,Y -141.711,Z 1259.152,A 0.000,B 0.000,C 90.000,E1 207.385} C_DIS
LIN {X 0.004,Y -139.472,Z 1259.116,A 0.000,B 0.000,C 90.000,E1 200.918} C_DIS
LIN {X -0.074,Y -139.204,Z 1259.106,A 0.000,B 0.000,C 90.000,E1 199.087} C_DIS
LIN {X -0.016,Y -138.329,Z 1259.054,A 0.000,B 0.000,C 90.000,E1 189.726} C_DIS
LIN {X -0.013,Y -139.440,Z 1259.007,A 0.000,B 0.000,C 90.000,E1 181.318} C_DIS
LIN {X 0.067,Y -140.972,Z 1258.976,A 0.000,B 0.000,C 90.000,E1 175.698} C_DIS
LIN {X 0.017,Y -142.728,Z 1258.956,A 0.000,B 0.000,C 90.000,E1 172.008} C_DIS
LIN {X -0.025,Y -145.113,Z 1258.930,A 0.000,B 0.000,C 90.000,E1 167.409} C_DIS
LIN {X -0.031,Y -147.737,Z 1258.910,A 0.000,B 0.000,C 90.000,E1 163.740} C_DIS
LIN {X 0.051,Y -150.401,Z 1258.889,A 0.000,B 0.000,C 90.000,E1 160.061} C_DIS
LIN {X -0.074,Y -153.837,Z 1258.869,A 0.000,B 0.000,C 90.000,E1 156.485} C_DIS
LIN {X -0.015,Y -157.248,Z 1258.849,A 0.000,B 0.000,C 90.000,E1 152.871} C_DIS
LIN {X -0.076,Y -161.421,Z 1258.829,A 0.000,B 0.000,C 90.000,E1 149.331} C_DIS
LIN {X -0.067,Y -165.621,Z 1258.810,A 0.000,B 0.000,C 90.000,E1 145.801} C_DIS
LIN {X 0.054,Y -170.550,Z 1258.791,A 0.000,B 0.000,C 90.000,E1 142.271} C_DIS
LIN {X -0.038,Y -175.429,Z 1258.771,A 0.000,B 0.000,C 90.000,E1 138.852} C_DIS
LIN {X 0.079,Y -181.053,Z 1258.752,A 0.000,B 0.000,C 90.000,E1 135.405} C_DIS
LIN {X -0.055,Y -186.488,Z 1258.734,A 0.000,B 0.000,C 90.000,E1 132.081} C_DIS
LIN {X 0.013,Y -191.110,Z 1258.720,A 0.000,B 0.000,C 90.000,E1 129.564} C_DIS
LIN {X -0.067,Y -196.904,Z 1258.702,A 0.000,B 0.000,C 90.000,E1 126.297} C_DIS
LIN {X 0.037,Y -200.219,Z 1258.692,A 0.000,B 0.000,C 90.000,E1 124.612} C_DIS
LIN {X 0.005,Y -310.006,Z 1258.692,A 0.000,B 0.000,C 90.000,E1 124.612} C_DIS
LIN {X -0.153,Y -311.699,Z 1258.692,A 0.000,B 0.000,C 90.000,E1 124.612} C_DIS
LIN {X -0.043,Y -315.856,Z 1258.691,A 0.000,B 0.000,C 90.000,E1 124.405} C_DIS
LIN {X 0.068,Y -318.221,Z 1258.690,A 0.000,B 0.000,C 90.000,E1 124.199} C_DIS
LIN {X 0.031,Y -321.449,Z 1258.688,A 0.000,B 0.000,C 90.000,E1 123.833} C_DIS
LIN {X 0.163,Y -323.373,Z 1258.686,A 0.000,B 0.000,C 90.000,E1 123.499} C_DIS
LIN {X 0.024,Y -324.870,Z 1258.685,A 0.000,B 0.000,C 90.000,E1 123.214} C_DIS
LIN {X -0.077,Y -339.211,Z 1258.664,A 0.000,B 0.000,C 90.000,E1 119.461} C_DIS
LIN {X 0.092,Y -351.475,Z 1258.648,A 0.000,B 0.000,C 90.000,E1 116.668} C_DIS
LIN {X 0.149,Y -365.230,Z 1258.633,A 0.000,B 0.000,C 90.000,E1 113.951} C_DIS
LIN {X 0.198,Y -378.798,Z 1258.620,A 0.000,B 0.000,C 90.000,E1 111.589} C_DIS
LIN {X -0.055,Y -393.728,Z 1258.607,A 0.000,B 0.000,C 90.000,E1 109.322} C_DIS
LIN {X 0.178,Y -410.128,Z 1258.595,A 0.000,B 0.000,C 90.000,E1 107.040} C_DIS
LIN {X -0.093,Y -428.110,Z 1258.583,A 0.000,B 0.000,C 90.000,E1 104.883} C_DIS
LIN {X -0.150,Y -447.651,Z 1258.571,A 0.000,B 0.000,C 90.000,E1 102.771} C_DIS
LIN {X 0.095,Y -467.914,Z 1258.560,A 0.000,B 0.000,C 90.000,E1 100.782} C_DIS
LIN {X 0.144,Y -475.463,Z 1258.556,A 0.000,B 0.000,C 90.000,E1 100.084} C_DIS
LIN {X 0.215,Y -477.291,Z 1258.555,A 0.000,B 0.000,C 90.000,E1 99.849} C_DIS
LIN {X 0.084,Y -478.828,Z 1258.553,A 0.000,B 0.000,C 90.000,E1 99.613} C_DIS
LIN {X -0.048,Y -479.976,Z 1258.552,A 0.000,B 0.000,C 90.000,E1 99.378} C_DIS
LIN {X 0.102,Y -481.352,Z 1258.549,A 0.000,B 0.000,C 90.000,E1 98.859} C_DIS
LIN {X -0.214,Y -481.696,Z 1258.547,A 0.000,B 0.000,C 90.000,E1 98.398} C_DIS
LIN {X 0.022,Y -481.067,Z 1258.544,A 0.000,B 0.000,C 90.000,E1 97.871} C_DIS
LIN {X 0.192,Y -479.363,Z 1258.541,A 0.000,B 0.000,C 90.000,E1 97.352} C_DIS
LIN {X 0.008,Y -478.012,Z 1258.540,A 0.000,B 0.000,C 90.000,E1 97.125} C_DIS
LIN {X 0.133,Y -456.224,Z 1258.523,A 0.000,B 0.000,C 90.000,E1 94.073} C_DIS
LIN {X -0.089,Y -435.756,Z 1258.505,A 0.000,B 0.000,C 90.000,E1 90.974} C_DIS
LIN {X 0.037,Y -420.519,Z 1258.490,A 0.000,B 0.000,C 90.000,E1 88.282} C_DIS
LIN {X 0.009,Y -409.046,Z 1258.478,A 0.000,B 0.000,C 90.000,E1 86.102} C_DIS
LIN {X 0.063,Y -400.414,Z 1258.469,A 0.000,B 0.000,C 90.000,E1 84.432} C_DIS
LIN {X 0.029,Y -390.182,Z 1258.458,A 0.000,B 0.000,C 90.000,E1 82.470} C_DIS
LIN {X 0.182,Y -381.260,Z 1258.449,A 0.000,B 0.000,C 90.000,E1 80.735} C_DIS
LIN {X -0.143,Y -372.069,Z 1258.439,A 0.000,B 0.000,C 90.000,E1 79.050} C_DIS
LIN {X -0.116,Y -362.519,Z 1258.429,A 0.000,B 0.000,C 90.000,E1 77.285} C_DIS
LIN {X 0.089,Y -352.777,Z 1258.419,A 0.000,B 0.000,C 90.000,E1 75.463} C_DIS
LIN {X -0.140,Y -341.327,Z 1258.407,A 0.000,B 0.000,C 90.000,E1 73.378} C_DIS
LIN {X 0.080,Y -326.828,Z 1258.392,A 0.000,B 0.000,C 90.000,E1 70.550} C_DIS
LIN {X -0.082,Y -313.088,Z 1258.376,A 0.000,B 0.000,C 90.000,E1 67.720} C_DIS
LIN {X 0.087,Y -297.708,Z 1258.356,A 0.000,B 0.000,C 90.000,E1 64.101} C_DIS
LIN {X -0.116,Y -285.262,Z 1258.338,A 0.000,B 0.000,C 90.000,E1 60.795} C_DIS
LIN {X -0.116,Y -273.982,Z 1258.319,A 0.000,B 0.000,C 90.000,E1 57.375} C_DIS
LIN {X 0.009,Y -263.722,Z 1258.299,A 0.000,B 0.000,C 90.000,E1 53.863} C_DIS
LIN {X -0.002,Y -254.363,Z 1258.280,A 0.000,B 0.000,C 90.000,E1 50.312} C_DIS
LIN {X -0.036,Y -245.616,Z 1258.259,A 0.000,B 0.000,C 90.000,E1 46.701} C_DIS
LIN {X -0.008,Y -237.413,Z 1258.239,A 0.000,B 0.000,C 90.000,E1 43.014} C_DIS
LIN {X 0.048,Y -231.119,Z 1258.222,A 0.000,B 0.000,C 90.000,E1 40.011} C_DIS
LIN {X 0.061,Y -223.756,Z 1258.201,A 0.000,B 0.000,C 90.000,E1 36.217} C_DIS
LIN {X -0.127,Y -217.070,Z 1258.180,A 0.000,B 0.000,C 90.000,E1 32.418} C_DIS
LIN {X -0.013,Y -211.062,Z 1258.158,A 0.000,B 0.000,C 90.000,E1 28.487} C_DIS
LIN {X 0.065,Y -205.968,Z 1258.136,A 0.000,B 0.000,C 90.000,E1 24.515} C_DIS
LIN {X -0.056,Y -201.598,Z 1258.114,A 0.000,B 0.000,C 90.000,E1 20.556} C_DIS
LIN {X -0.060,Y -197.325,Z 1258.087,A 0.000,B 0.000,C 90.000,E1 15.717} C_DIS
LIN {X -0.061,Y -193.768,Z 1258.056,A 0.000,B 0.000,C 90.000,E1 10.018} C_DIS
LIN {X 0.057,Y -194.660,Z 1257.956,A 0.000,B 0.000,C 90.000,E1 352.129} C_DIS
LIN {X 0.077,Y -197.861,Z 1257.929,A 0.000,B 0.000,C 90.000,E1 347.229} C_DIS
LIN {X -0.081,Y -202.129,Z 1257.902,A 0.000,B 0.000,C 90.000,E1 342.417} C_DIS
LIN {X -0.103,Y -206.416,Z 1257.880,A 0.000,B 0.000,C 90.000,E1 338.411} C_DIS
LIN {X 0.005,Y -211.475,Z 1257.858,A 0.000,B 0.000,C 90.000,E1 334.409} C_DIS
LIN {X 0.076,Y -217.112,Z 1257.836,A 0.000,B 0.000,C 90.000,E1 330.461} C_DIS
LIN {X -0.106,Y -223.536,Z 1257.814,A 0.000,B 0.000,C 90.000,E1 326.628} C_DIS
LIN {X 0.040,Y -230.689,Z 1257.793,A 0.000,B 0.000,C 90.000,E1 322.763} C_DIS
LIN {X -0.041,Y -238.682,Z 1257.772,A 0.000,B 0.000,C 90.000,E1 319.013} C_DIS
LIN {X -0.121,Y -247.641,Z 1257.752,A 0.000,B 0.000,C 90.000,E1 315.324} C_DIS
LIN {X 0.069,Y -255.771,Z 1257.735,A 0.000,B 0.000,C 90.000,E1 312.366} C_DIS
LIN {X -0.059,Y -263.980,Z 1257.722,A 0.000,B 0.000,C 90.000,E1 309.886} C_DIS
LIN {X 0.125,Y -271.988,Z 1257.710,A 0.000,B 0.000,C 90.000,E1 307.729} C_DIS
LIN {X -0.035,Y -281.043,Z 1257.698,A 0.000,B 0.000,C 90.000,E1 305.678} C_DIS
LIN {X -0.063,Y -294.661,Z 1257.683,A 0.000,B 0.000,C 90.000,E1 302.959} C_DIS
LIN {X 0.107,Y -304.170,Z 1257.674,A 0.000,B 0.000,C 90.000,E1 301.258} C_DIS
LIN {X 0.076,Y -312.636,Z 1257.667,A 0.000,B 0.000,C 90.000,E1 299.951} C_DIS
LIN {X 0.038,Y -326.721,Z 1257.656,A 0.000,B 0.000,C 90.000,E1 298.025} C_DIS
LIN {X -0.034,Y -347.004,Z 1257.642,A 0.000,B 0.000,C 90.000,E1 295.540} C_DIS
LIN {X -0.008,Y -360.173,Z 1257.633,A 0.000,B 0.000,C 90.000,E1 294.027} C_DIS
LIN {X 0.016,Y -375.646,Z 1257.624,A 0.000,B 0.000,C 90.000,E1 292.280} C_DIS
LIN {X -0.036,Y -388.439,Z 1257.616,A 0.000,B 0.000,C 90.000,E1 290.844} C_DIS
LIN {X 0.024,Y -409.017,Z 1257.603,A 0.000,B 0.000,C 90.000,E1 288.598} C_DIS
LIN {X 0.176,Y -419.070,Z 1257.597,A 0.000,B 0.000,C 90.000,E1 287.511} C_DIS
LIN {X -0.081,Y -426.409,Z 1257.593,A 0.000,B 0.000,C 90.000,E1 286.732} C_DIS
LIN {X 0.099,Y -433.266,Z 1257.588,A 0.000,B 0.000,C 90.000,E1 285.898} C_DIS
LIN {X -0.186,Y -439.589,Z 1257.584,A 0.000,B 0.000,C 90.000,E1 285.134} C_DIS
LIN {X 0.121,Y -445.292,Z 1257.580,A 0.000,B 0.000,C 90.000,E1 284.300} C_DIS
LIN {X -0.056,Y -450.339,Z 1257.575,A 0.000,B 0.000,C 90.000,E1 283.536} C_DIS
LIN {X -0.194,Y -454.692,Z 1257.571,A 0.000,B 0.000,C 90.000,E1 282.771} C_DIS
LIN {X 0.157,Y -458.332,Z 1257.567,A 0.000,B 0.000,C 90.000,E1 281.951} C_DIS
LIN {X 0.090,Y -461.332,Z 1257.562,A 0.000,B 0.000,C 90.000,E1 281.186} C_DIS
LIN {X 0.204,Y -463.002,Z 1257.559,A 0.000,B 0.000,C 90.000,E1 280.658} C_DIS
LIN {X -0.211,Y -464.400,Z 1257.557,A 0.000,B 0.000,C 90.000,E1 280.197} C_DIS
LIN {X -0.079,Y -465.548,Z 1257.554,A 0.000,B 0.000,C 90.000,E1 279.670} C_DIS
LIN {X -0.015,Y -466.391,Z 1257.551,A 0.000,B 0.000,C 90.000,E1 279.151} C_DIS
LIN {X 0.129,Y -466.900,Z 1257.548,A 0.000,B 0.000,C 90.000,E1 278.624} C_DIS
LIN {X 0.207,Y -467.056,Z 1257.545,A 0.000,B 0.000,C 90.000,E1 278.106} C_DIS
LIN {X -0.173,Y -466.778,Z 1257.542,A 0.000,B 0.000,C 90.000,E1 277.644} C_DIS
LIN {X -0.087,Y -466.077,Z 1257.540,A 0.000,B 0.000,C 90.000,E1 277.125} C_DIS
LIN {X -0.003,Y -464.959,Z 1257.537,A 0.000,B 0.000,C 90.000,E1 276.606} C_DIS
LIN {X 0.077,Y -463.403,Z 1257.534,A 0.000,B 0.000,C 90.000,E1 276.087} C_DIS
LIN {X -0.026,Y -460.422,Z 1257.530,A 0.000,B 0.000,C 90.000,E1 275.334} C_DIS
LIN {X -0.014,Y -458.013,Z 1257.527,A 0.000,B 0.000,C 90.000,E1 274.821} C_DIS
LIN {X 0.024,Y -454.957,Z 1257.524,A 0.000,B 0.000,C 90.000,E1 274.302} C_DIS
LIN {X 0.043,Y -451.216,Z 1257.521,A 0.000,B 0.000,C 90.000,E1 273.784} C_DIS
LIN {X -0.191,Y -448.980,Z 1257.520,A 0.000,B 0.000,C 90.000,E1 273.555} C_DIS
LIN {X 0.014,Y -446.421,Z 1257.518,A 0.000,B 0.000,C 90.000,E1 273.269} C_DIS
LIN {X -0.202,Y -443.534,Z 1257.517,A 0.000,B 0.000,C 90.000,E1 273.037} C_DIS
LIN {X 0.183,Y -440.580,Z 1257.515,A 0.000,B 0.000,C 90.000,E1 272.751} C_DIS
LIN {X -0.082,Y -434.121,Z 1257.513,A 0.000,B 0.000,C 90.000,E1 272.350} C_DIS
LIN {X 0.198,Y -427.241,Z 1257.511,A 0.000,B 0.000,C 90.000,E1 271.949} C_DIS
LIN {X 0.080,Y -420.291,Z 1257.509,A 0.000,B 0.000,C 90.000,E1 271.661} C_DIS
LIN {X -0.111,Y -413.154,Z 1257.508,A 0.000,B 0.000,C 90.000,E1 271.432} C_DIS
LIN {X 0.012,Y -406.110,Z 1257.507,A 0.000,B 0.000,C 90.000,E1 271.203} C_DIS
LIN {X -0.035,Y -398.880,Z 1257.506,A 0.000,B 0.000,C 90.000,E1 271.031} C_DIS
LIN {X 0.122,Y -391.409,Z 1257.505,A 0.000,B 0.000,C 90.000,E1 270.859} C_DIS
LIN {X 0.084,Y -382.771,Z 1257.504,A 0.000,B 0.000,C 90.000,E1 270.745} C_DIS
LIN {X 0.078,Y -368.887,Z 1257.504,A 0.000,B 0.000,C 90.000,E1 270.630} C_DIS
LIN {X -0.052,Y -361.271,Z 1257.503,A 0.000,B 0.000,C 90.000,E1 270.630} C_DIS
LIN {X -0.062,Y -181.546,Z 1257.503,A 0.000,B 0.000,C 90.000,E1 270.630} C_DIS
LIN {X -0.058,Y -181.295,Z 1257.494,A 0.000,B 0.000,C 90.000,E1 268.912} C_DIS
LIN {X -0.008,Y -180.908,Z 1257.475,A 0.000,B 0.000,C 90.000,E1 265.527} C_DIS
LIN {X 0.049,Y -180.759,Z 1257.470,A 0.000,B 0.000,C 90.000,E1 264.666} C_DIS
LIN {X -0.059,Y -178.853,Z 1257.442,A 0.000,B 0.000,C 90.000,E1 259.634} C_DIS
LIN {X 0.012,Y -175.897,Z 1257.414,A 0.000,B 0.000,C 90.000,E1 254.519} C_DIS
LIN {X -0.049,Y -174.572,Z 1257.405,A 0.000,B 0.000,C 90.000,E1 252.834} C_DIS
LIN {X -0.013,Y -171.555,Z 1257.381,A 0.000,B 0.000,C 90.000,E1 248.539} C_DIS
LIN {X 0.042,Y -167.779,Z 1257.357,A 0.000,B 0.000,C 90.000,E1 244.204} C_DIS
LIN {X -0.016,Y -166.492,Z 1257.347,A 0.000,B 0.000,C 90.000,E1 242.487} C_DIS
LIN {X -0.020,Y -163.202,Z 1257.328,A 0.000,B 0.000,C 90.000,E1 238.997} C_DIS
LIN {X 0.034,Y -161.166,Z 1257.313,A 0.000,B 0.000,C 90.000,E1 236.342} C_DIS
LIN {X 0.069,Y -157.182,Z 1257.288,A 0.000,B 0.000,C 90.000,E1 231.904} C_DIS
LIN {X -0.008,Y -155.912,Z 1257.279,A 0.000,B 0.000,C 90.000,E1 230.150} C_DIS
LIN {X 0.048,Y -152.162,Z 1257.254,A 0.000,B 0.000,C 90.000,E1 225.648} C_DIS
LIN {X 0.068,Y -150.411,Z 1257.239,A 0.000,B 0.000,C 90.000,E1 222.933} C_DIS
LIN {X 0.000,Y -147.140,Z 1257.213,A 0.000,B 0.000,C 90.000,E1 218.418} C_DIS
LIN {X -0.003,Y -145.699,Z 1257.198,A 0.000,B 0.000,C 90.000,E1 215.678} C_DIS
LIN {X 0.005,Y -143.083,Z 1257.173,A 0.000,B 0.000,C 90.000,E1 211.082} C_DIS
LIN {X 0.010,Y -141.700,Z 1257.152,A 0.000,B 0.000,C 90.000,E1 207.385} C_DIS
LIN {X -0.068,Y -139.466,Z 1257.116,A 0.000,B 0.000,C 90.000,E1 200.918} C_DIS
LIN {X -0.014,Y -139.200,Z 1257.106,A 0.000,B 0.000,C 90.000,E1 199.033} C_DIS
LIN {X 0.050,Y -138.328,Z 1257.054,A 0.000,B 0.000,C 90.000,E1 189.670} C_DIS
LIN {X 0.055,Y -139.445,Z 1257.007,A 0.000,B 0.000,C 90.000,E1 181.260} C_DIS
LIN {X -0.004,Y -140.985,Z 1256.976,A 0.000,B 0.000,C 90.000,E1 175.698} C_DIS
LIN {X -0.055,Y -142.739,Z 1256.955,A 0.000,B 0.000,C 90.000,E1 172.008} C_DIS
LIN {X 0.043,Y -145.132,Z 1256.930,A 0.000,B 0.000,C 90.000,E1 167.353} C_DIS
LIN {X 0.037,Y -147.755,Z 1256.909,A 0.000,B 0.000,C 90.000,E1 163.685} C_DIS
LIN {X -0.023,Y -150.425,Z 1256.889,A 0.000,B 0.000,C 90.000,E1 160.061} C_DIS
LIN {X -0.009,Y -153.867,Z 1256.869,A 0.000,B 0.000,C 90.000,E1 156.433} C_DIS
LIN {X 0.047,Y -157.277,Z 1256.849,A 0.000,B 0.000,C 90.000,E1 152.820} C_DIS
LIN {X -0.015,Y -161.457,Z 1256.829,A 0.000,B 0.000,C 90.000,E1 149.282} C_DIS
LIN {X -0.008,Y -165.657,Z 1256.810,A 0.000,B 0.000,C 90.000,E1 145.754} C_DIS
LIN {X -0.028,Y -170.593,Z 1256.790,A 0.000,B 0.000,C 90.000,E1 142.271} C_DIS
LIN {X 0.012,Y -175.469,Z 1256.771,A 0.000,B 0.000,C 90.000,E1 138.809} C_DIS
LIN {X -0.006,Y -181.092,Z 1256.752,A 0.000,B 0.000,C 90.000,E1 135.405} C_DIS
LIN {X -0.016,Y -186.534,Z 1256.734,A 0.000,B 0.000,C 90.000,E1 132.043} C_DIS
LIN {X -0.074,Y -191.151,Z 1256.720,A 0.000,B 0.000,C 90.000,E1 129.564} C_DIS
LIN {X 0.003,Y -196.953,Z 1256.701,A 0.000,B 0.000,C 90.000,E1 126.251} C_DIS
LIN {X -0.029,Y -200.259,Z 1256.692,A 0.000,B 0.000,C 90.000,E1 124.612} C_DIS
LIN {X -0.080,Y -309.279,Z 1256.692,A 0.000,B 0.000,C 90.000,E1 124.612} C_DIS
LIN {X 0.142,Y -311.941,Z 1256.692,A 0.000,B 0.000,C 90.000,E1 124.532} C_DIS
LIN {X -0.184,Y -315.978,Z 1256.691,A 0.000,B 0.000,C 90.000,E1 124.405} C_DIS
LIN {X -0.072,Y -318.320,Z 1256.690,A 0.000,B 0.000,C 90.000,E1 124.199} C_DIS
LIN {X 0.155,Y -321.530,Z 1256.688,A 0.000,B 0.000,C 90.000,E1 123.785} C_DIS
LIN {X 0.012,Y -323.454,Z 1256.686,A 0.000,B 0.000,C 90.000,E1 123.499} C_DIS
LIN {X 0.139,Y -324.951,Z 1256.684,A 0.000,B 0.000,C 90.000,E1 123.166} C_DIS
LIN {X -0.079,Y -338.021,Z 1256.665,A 0.000,B 0.000,C 90.000,E1 119.745} C_DIS
LIN {X 0.064,Y -350.146,Z 1256.650,A 0.000,B 0.000,C 90.000,E1 116.950} C_DIS
LIN {X -0.082,Y -363.740,Z 1256.635,A 0.000,B 0.000,C 90.000,E1 114.259} C_DIS
LIN {X -0.081,Y -377.158,Z 1256.622,A 0.000,B 0.000,C 90.000,E1 111.897} C_DIS
LIN {X -0.014,Y -391.928,Z 1256.609,A 0.000,B 0.000,C 90.000,E1 109.577} C_DIS
LIN {X -0.084,Y -408.153,Z 1256.596,A 0.000,B 0.000,C 90.000,E1 107.330} C_DIS
LIN {X -0.121,Y -425.949,Z 1256.584,A 0.000,B 0.000,C 90.000,E1 105.134} C_DIS
LIN {X -0.159,Y -445.339,Z 1256.572,A 0.000,B 0.000,C 90.000,E1 103.008} C_DIS
LIN {X 0.018,Y -465.540,Z 1256.561,A 0.000,B 0.000,C 90.000,E1 101.007} C_DIS
LIN {X -0.016,Y -473.269,Z 1256.557,A 0.000,B 0.000,C 90.000,E1 100.310} C_DIS
LIN {X 0.055,Y -475.599,Z 1256.556,A 0.000,B 0.000,C 90.000,E1 100.074} C_DIS
LIN {X 0.044,Y -477.362,Z 1256.555,A 0.000,B 0.000,C 90.000,E1 99.849} C_DIS
LIN {X -0.086,Y -478.847,Z 1256.553,A 0.000,B 0.000,C 90.000,E1 99.613} C_DIS
LIN {X 0.255,Y -479.953,Z 1256.552,A 0.000,B 0.000,C 90.000,E1 99.321} C_DIS
LIN {X -0.069,Y -481.264,Z 1256.549,A 0.000,B 0.000,C 90.000,E1 98.859} C_DIS
LIN {X 0.091,Y -481.552,Z 1256.546,A 0.000,B 0.000,C 90.000,E1 98.341} C_DIS
LIN {X -0.149,Y -480.864,Z 1256.544,A 0.000,B 0.000,C 90.000,E1 97.871} C_DIS
LIN {X 0.020,Y -479.091,Z 1256.541,A 0.000,B 0.000,C 90.000,E1 97.352} C_DIS
LIN {X -0.164,Y -477.693,Z 1256.539,A 0.000,B 0.000,C 90.000,E1 97.125} C_DIS
LIN {X -0.042,Y -455.879,Z 1256.523,A 0.000,B 0.000,C 90.000,E1 94.073} C_DIS
LIN {X 0.168,Y -435.436,Z 1256.505,A 0.000,B 0.000,C 90.000,E1 90.917} C_DIS
LIN {X -0.016,Y -418.732,Z 1256.489,A 0.000,B 0.000,C 90.000,E1 87.993} C_DIS
LIN {X -0.175,Y -408.724,Z 1256.478,A 0.000,B 0.000,C 90.000,E1 86.102} C_DIS
LIN {X -0.080,Y -398.641,Z 1256.467,A 0.000,B 0.000,C 90.000,E1 84.147} C_DIS
LIN {X -0.158,Y -388.385,Z 1256.456,A 0.000,B 0.000,C 90.000,E1 82.186} C_DIS
LIN {X 0.020,Y -379.428,Z 1256.447,A 0.000,B 0.000,C 90.000,E1 80.443} C_DIS
LIN {X 0.032,Y -371.753,Z 1256.439,A 0.000,B 0.000,C 90.000,E1 78.993} C_DIS
LIN {X 0.047,Y -362.201,Z 1256.429,A 0.000,B 0.000,C 90.000,E1 77.229} C_DIS
LIN {X -0.104,Y -352.465,Z 1256.419,A 0.000,B 0.000,C 90.000,E1 75.463} C_DIS
LIN {X -0.004,Y -341.022,Z 1256.407,A 0.000,B 0.000,C 90.000,E1 73.323} C_DIS
LIN {X -0.112,Y -326.572,Z 1256.392,A 0.000,B 0.000,C 90.000,E1 70.550} C_DIS
LIN {X -0.055,Y -311.377,Z 1256.374,A 0.000,B 0.000,C 90.000,E1 67.358} C_DIS
LIN {X 0.027,Y -297.500,Z 1256.356,A 0.000,B 0.000,C 90.000,E1 64.076} C_DIS
LIN {X 0.084,Y -285.039,Z 1256.337,A 0.000,B 0.000,C 90.000,E1 60.717} C_DIS
LIN {X -0.072,Y -273.715,Z 1256.318,A 0.000,B 0.000,C 90.000,E1 57.327} C_DIS
LIN {X -0.031,Y -263.414,Z 1256.299,A 0.000,B 0.000,C 90.000,E1 53.829} C_DIS
LIN {X -0.037,Y -254.023,Z 1256.279,A 0.000,B 0.000,C 90.000,E1 50.275} C_DIS
LIN {X 0.109,Y -245.269,Z 1256.259,A 0.000,B 0.000,C 90.000,E1 46.620} C_DIS
LIN {X -0.053,Y -237.041,Z 1256.239,A 0.000,B 0.000,C 90.000,E1 42.975} C_DIS
LIN {X 0.081,Y -229.197,Z 1256.218,A 0.000,B 0.000,C 90.000,E1 39.197} C_DIS
LIN {X 0.080,Y -221.944,Z 1256.197,A 0.000,B 0.000,C 90.000,E1 35.391} C_DIS
LIN {X 0.021,Y -215.350,Z 1256.175,A 0.000,B 0.000,C 90.000,E1 31.544} C_DIS
LIN {X -0.027,Y -209.486,Z 1256.154,A 0.000,B 0.000,C 90.000,E1 27.641} C_DIS
LIN {X 0.099,Y -204.550,Z 1256.131,A 0.000,B 0.000,C 90.000,E1 23.643} C_DIS
LIN {X -0.068,Y -200.352,Z 1256.109,A 0.000,B 0.000,C 90.000,E1 19.685} C_DIS
LIN {X -0.055,Y -196.264,Z 1256.082,A 0.000,B 0.000,C 90.000,E1 14.828} C_DIS
LIN {X 0.016,Y -193.021,Z 1256.051,A 0.000,B 0.000,C 90.000,E1 9.095} C_DIS
LIN {X 0.098,Y -194.009,Z 1255.961,A 0.000,B 0.000,C 90.000,E1 352.932} C_DIS
LIN {X 0.055,Y -197.664,Z 1255.929,A 0.000,B 0.000,C 90.000,E1 347.229} C_DIS
LIN {X 0.082,Y -201.966,Z 1255.902,A 0.000,B 0.000,C 90.000,E1 342.362} C_DIS
LIN {X 0.052,Y -206.282,Z 1255.880,A 0.000,B 0.000,C 90.000,E1 338.358} C_DIS
LIN {X -0.036,Y -211.361,Z 1255.858,A 0.000,B 0.000,C 90.000,E1 334.409} C_DIS
LIN {X 0.031,Y -217.022,Z 1255.836,A 0.000,B 0.000,C 90.000,E1 330.461} C_DIS
LIN {X 0.032,Y -223.477,Z 1255.814,A 0.000,B 0.000,C 90.000,E1 326.580} C_DIS
LIN {X -0.012,Y -230.625,Z 1255.793,A 0.000,B 0.000,C 90.000,E1 322.763} C_DIS
LIN {X -0.097,Y -238.624,Z 1255.772,A 0.000,B 0.000,C 90.000,E1 319.013} C_DIS
LIN {X -0.006,Y -247.577,Z 1255.752,A 0.000,B 0.000,C 90.000,E1 315.283} C_DIS
LIN {X 0.005,Y -255.719,Z 1255.735,A 0.000,B 0.000,C 90.000,E1 312.366} C_DIS
LIN {X 0.042,Y -263.921,Z 1255.721,A 0.000,B 0.000,C 90.000,E1 309.850} C_DIS
LIN {X 0.054,Y -271.935,Z 1255.710,A 0.000,B 0.000,C 90.000,E1 307.729} C_DIS
LIN {X -0.051,Y -279.430,Z 1255.700,A 0.000,B 0.000,C 90.000,E1 306.011} C_DIS
LIN {X 0.138,Y -291.068,Z 1255.687,A 0.000,B 0.000,C 90.000,E1 303.579} C_DIS
LIN {X 0.002,Y -300.166,Z 1255.677,A 0.000,B 0.000,C 90.000,E1 301.926} C_DIS
LIN {X 0.072,Y -308.188,Z 1255.670,A 0.000,B 0.000,C 90.000,E1 300.590} C_DIS
LIN {X 0.159,Y -319.397,Z 1255.661,A 0.000,B 0.000,C 90.000,E1 298.949} C_DIS
LIN {X 0.154,Y -341.695,Z 1255.645,A 0.000,B 0.000,C 90.000,E1 296.104} C_DIS
LIN {X -0.200,Y -357.520,Z 1255.635,A 0.000,B 0.000,C 90.000,E1 294.335} C_DIS
LIN {X 0.045,Y -370.597,Z 1255.627,A 0.000,B 0.000,C 90.000,E1 292.823} C_DIS
LIN {X -0.154,Y -383.461,Z 1255.619,A 0.000,B 0.000,C 90.000,E1 291.408} C_DIS
LIN {X 0.150,Y -401.262,Z 1255.608,A 0.000,B 0.000,C 90.000,E1 289.396} C_DIS
LIN {X -0.196,Y -416.633,Z 1255.599,A 0.000,B 0.000,C 90.000,E1 287.819} C_DIS
LIN {X -0.013,Y -424.046,Z 1255.594,A 0.000,B 0.000,C 90.000,E1 286.985} C_DIS
LIN {X 0.026,Y -433.310,Z 1255.588,A 0.000,B 0.000,C 90.000,E1 285.898} C_DIS
LIN {X -0.260,Y -439.621,Z 1255.584,A 0.000,B 0.000,C 90.000,E1 285.134} C_DIS
LIN {X 0.046,Y -445.326,Z 1255.579,A 0.000,B 0.000,C 90.000,E1 284.300} C_DIS
LIN {X -0.130,Y -450.331,Z 1255.575,A 0.000,B 0.000,C 90.000,E1 283.536} C_DIS
LIN {X 0.174,Y -454.693,Z 1255.571,A 0.000,B 0.000,C 90.000,E1 282.715} C_DIS
LIN {X 0.082,Y -458.340,Z 1255.566,A 0.000,B 0.000,C 90.000,E1 281.951} C_DIS
LIN {X 0.014,Y -461.325,Z 1255.562,A 0.000,B 0.000,C 90.000,E1 281.186} C_DIS
LIN {X 0.128,Y -463.004,Z 1255.559,A 0.000,B 0.000,C 90.000,E1 280.658} C_DIS
LIN {X 0.169,Y -464.406,Z 1255.556,A 0.000,B 0.000,C 90.000,E1 280.141} C_DIS
LIN {X -0.156,Y -465.536,Z 1255.554,A 0.000,B 0.000,C 90.000,E1 279.670} C_DIS
LIN {X -0.092,Y -466.378,Z 1255.551,A 0.000,B 0.000,C 90.000,E1 279.151} C_DIS
LIN {X 0.052,Y -466.931,Z 1255.548,A 0.000,B 0.000,C 90.000,E1 278.624} C_DIS
LIN {X 0.130,Y -467.118,Z 1255.545,A 0.000,B 0.000,C 90.000,E1 278.106} C_DIS
LIN {X 0.213,Y -466.851,Z 1255.542,A 0.000,B 0.000,C 90.000,E1 277.587} C_DIS
LIN {X -0.164,Y -466.216,Z 1255.539,A 0.000,B 0.000,C 90.000,E1 277.125} C_DIS
LIN {X -0.080,Y -465.086,Z 1255.537,A 0.000,B 0.000,C 90.000,E1 276.606} C_DIS
LIN {X 0.002,Y -463.576,Z 1255.534,A 0.000,B 0.000,C 90.000,E1 276.087} C_DIS
LIN {X -0.100,Y -460.615,Z 1255.530,A 0.000,B 0.000,C 90.000,E1 275.334} C_DIS
LIN {X -0.085,Y -458.192,Z 1255.527,A 0.000,B 0.000,C 90.000,E1 274.821} C_DIS
LIN {X -0.046,Y -455.157,Z 1255.524,A 0.000,B 0.000,C 90.000,E1 274.302} C_DIS
LIN {X 0.210,Y -453.434,Z 1255.522,A 0.000,B 0.000,C 90.000,E1 274.012} C_DIS
LIN {X 0.190,Y -449.210,Z 1255.520,A 0.000,B 0.000,C 90.000,E1 273.498} C_DIS
LIN {X -0.054,Y -446.701,Z 1255.518,A 0.000,B 0.000,C 90.000,E1 273.269} C_DIS
LIN {X 0.175,Y -443.822,Z 1255.517,A 0.000,B 0.000,C 90.000,E1 272.980} C_DIS
LIN {X 0.058,Y -437.626,Z 1255.514,A 0.000,B 0.000,C 90.000,E1 272.522} C_DIS
LIN {X -0.012,Y -430.690,Z 1255.512,A 0.000,B 0.000,C 90.000,E1 272.121} C_DIS
LIN {X 0.105,Y -423.802,Z 1255.510,A 0.000,B 0.000,C 90.000,E1 271.776} C_DIS
LIN {X 0.151,Y -416.661,Z 1255.508,A 0.000,B 0.000,C 90.000,E1 271.489} C_DIS
LIN {X -0.144,Y -406.168,Z 1255.507,A 0.000,B 0.000,C 90.000,E1 271.203} C_DIS
LIN {X -0.179,Y -398.937,Z 1255.506,A 0.000,B 0.000,C 90.000,E1 271.031} C_DIS
LIN {X -0.017,Y -391.541,Z 1255.505,A 0.000,B 0.000,C 90.000,E1 270.859} C_DIS
LIN {X -0.017,Y -377.987,Z 1255.504,A 0.000,B 0.000,C 90.000,E1 270.688} C_DIS
LIN {X -0.124,Y -364.748,Z 1255.503,A 0.000,B 0.000,C 90.000,E1 270.630} C_DIS
LIN {X 0.087,Y -181.548,Z 1255.503,A 0.000,B 0.000,C 90.000,E1 270.573} C_DIS
LIN {X -0.052,Y -181.460,Z 1255.498,A 0.000,B 0.000,C 90.000,E1 269.599} C_DIS
LIN {X 0.081,Y -180.896,Z 1255.473,A 0.000,B 0.000,C 90.000,E1 265.179} C_DIS
LIN {X -0.091,Y -179.842,Z 1255.459,A 0.000,B 0.000,C 90.000,E1 262.704} C_DIS
LIN {X -0.034,Y -179.026,Z 1255.445,A 0.000,B 0.000,C 90.000,E1 260.151} C_DIS
LIN {X 0.028,Y -178.672,Z 1255.441,A 0.000,B 0.000,C 90.000,E1 259.285} C_DIS
LIN {X -0.036,Y -175.722,Z 1255.412,A 0.000,B 0.000,C 90.000,E1 254.212} C_DIS
LIN {X -0.020,Y -172.437,Z 1255.388,A 0.000,B 0.000,C 90.000,E1 249.934} C_DIS
LIN {X -0.065,Y -171.268,Z 1255.379,A 0.000,B 0.000,C 90.000,E1 248.230} C_DIS
LIN {X -0.018,Y -167.538,Z 1255.355,A 0.000,B 0.000,C 90.000,E1 243.896} C_DIS
LIN {X -0.004,Y -166.153,Z 1255.345,A 0.000,B 0.000,C 90.000,E1 242.153} C_DIS
LIN {X -0.013,Y -162.930,Z 1255.326,A 0.000,B 0.000,C 90.000,E1 238.663} C_DIS
LIN {X -0.036,Y -161.602,Z 1255.316,A 0.000,B 0.000,C 90.000,E1 236.914} C_DIS
LIN {X -0.060,Y -159.125,Z 1255.301,A 0.000,B 0.000,C 90.000,E1 234.276} C_DIS
LIN {X -0.049,Y -155.648,Z 1255.277,A 0.000,B 0.000,C 90.000,E1 229.828} C_DIS
LIN {X 0.004,Y -151.919,Z 1255.252,A 0.000,B 0.000,C 90.000,E1 225.324} C_DIS
LIN {X 0.019,Y -150.154,Z 1255.237,A 0.000,B 0.000,C 90.000,E1 222.609} C_DIS
LIN {X -0.060,Y -146.935,Z 1255.212,A 0.000,B 0.000,C 90.000,E1 218.096} C_DIS
LIN {X 0.046,Y -145.524,Z 1255.196,A 0.000,B 0.000,C 90.000,E1 215.311} C_DIS
LIN {X 0.040,Y -142.923,Z 1255.171,A 0.000,B 0.000,C 90.000,E1 210.718} C_DIS
LIN {X -0.033,Y -141.546,Z 1255.150,A 0.000,B 0.000,C 90.000,E1 207.052} C_DIS
LIN {X -0.044,Y -139.404,Z 1255.114,A 0.000,B 0.000,C 90.000,E1 200.556} C_DIS
LIN {X 0.010,Y -139.122,Z 1255.104,A 0.000,B 0.000,C 90.000,E1 198.671} C_DIS
LIN {X 0.041,Y -138.352,Z 1255.057,A 0.000,B 0.000,C 90.000,E1 190.254} C_DIS
LIN {X 0.032,Y -139.502,Z 1255.005,A 0.000,B 0.000,C 90.000,E1 180.917} C_DIS
LIN {X -0.028,Y -141.133,Z 1254.974,A 0.000,B 0.000,C 90.000,E1 175.355} C_DIS
LIN {X -0.075,Y -142.514,Z 1254.959,A 0.000,B 0.000,C 90.000,E1 172.591} C_DIS
LIN {X 0.012,Y -144.773,Z 1254.933,A 0.000,B 0.000,C 90.000,E1 167.937} C_DIS
LIN {X -0.039,Y -147.387,Z 1254.913,A 0.000,B 0.000,C 90.000,E1 164.283} C_DIS
LIN {X 0.024,Y -150.717,Z 1254.887,A 0.000,B 0.000,C 90.000,E1 159.699} C_DIS
LIN {X -0.036,Y -154.198,Z 1254.867,A 0.000,B 0.000,C 90.000,E1 156.102} C_DIS
LIN {X 0.034,Y -157.637,Z 1254.847,A 0.000,B 0.000,C 90.000,E1 152.487} C_DIS
LIN {X -0.019,Y -161.896,Z 1254.827,A 0.000,B 0.000,C 90.000,E1 148.948} C_DIS
LIN {X 0.090,Y -166.086,Z 1254.808,A 0.000,B 0.000,C 90.000,E1 145.388} C_DIS
LIN {X 0.088,Y -171.094,Z 1254.789,A 0.000,B 0.000,C 90.000,E1 141.904} C_DIS
LIN {X 0.009,Y -175.968,Z 1254.769,A 0.000,B 0.000,C 90.000,E1 138.485} C_DIS
LIN {X 0.122,Y -180.213,Z 1254.755,A 0.000,B 0.000,C 90.000,E1 135.891} C_DIS
LIN {X 0.097,Y -185.628,Z 1254.736,A 0.000,B 0.000,C 90.000,E1 132.528} C_DIS
LIN {X -0.117,Y -190.224,Z 1254.723,A 0.000,B 0.000,C 90.000,E1 130.092} C_DIS
LIN {X 0.042,Y -197.552,Z 1254.700,A 0.000,B 0.000,C 90.000,E1 125.931} C_DIS
LIN {X -0.109,Y -200.306,Z 1254.692,A 0.000,B 0.000,C 90.000,E1 124.612} C_DIS
LIN {X 0.046,Y -309.943,Z 1254.692,A 0.000,B 0.000,C 90.000,E1 124.565} C_DIS
LIN {X 0.096,Y -311.485,Z 1254.692,A 0.000,B 0.000,C 90.000,E1 124.532} C_DIS
LIN {X -0.052,Y -316.536,Z 1254.691,A 0.000,B 0.000,C 90.000,E1 124.326} C_DIS
LIN {X -0.057,Y -319.701,Z 1254.689,A 0.000,B 0.000,C 90.000,E1 124.040} C_DIS
LIN {X 0.068,Y -323.339,Z 1254.686,A 0.000,B 0.000,C 90.000,E1 123.499} C_DIS
LIN {X 0.148,Y -324.905,Z 1254.684,A 0.000,B 0.000,C 90.000,E1 123.166} C_DIS
LIN {X 0.059,Y -339.278,Z 1254.663,A 0.000,B 0.000,C 90.000,E1 119.411} C_DIS
LIN {X -0.075,Y -351.560,Z 1254.648,A 0.000,B 0.000,C 90.000,E1 116.668} C_DIS
LIN {X -0.018,Y -365.324,Z 1254.633,A 0.000,B 0.000,C 90.000,E1 113.951} C_DIS
LIN {X 0.028,Y -378.906,Z 1254.620,A 0.000,B 0.000,C 90.000,E1 111.589} C_DIS
LIN {X 0.143,Y -393.852,Z 1254.607,A 0.000,B 0.000,C 90.000,E1 109.268} C_DIS
LIN {X 0.002,Y -410.267,Z 1254.595,A 0.000,B 0.000,C 90.000,E1 107.040} C_DIS
LIN {X 0.140,Y -428.267,Z 1254.583,A 0.000,B 0.000,C 90.000,E1 104.828} C_DIS
LIN {X 0.108,Y -447.817,Z 1254.571,A 0.000,B 0.000,C 90.000,E1 102.715} C_DIS
LIN {X -0.078,Y -468.086,Z 1254.560,A 0.000,B 0.000,C 90.000,E1 100.782} C_DIS
LIN {X -0.015,Y -473.237,Z 1254.557,A 0.000,B 0.000,C 90.000,E1 100.310} C_DIS
LIN {X 0.036,Y -475.566,Z 1254.556,A 0.000,B 0.000,C 90.000,E1 100.074} C_DIS
LIN {X -0.118,Y -477.420,Z 1254.555,A 0.000,B 0.000,C 90.000,E1 99.849} C_DIS
LIN {X -0.191,Y -478.824,Z 1254.553,A 0.000,B 0.000,C 90.000,E1 99.613} C_DIS
LIN {X -0.049,Y -480.669,Z 1254.551,A 0.000,B 0.000,C 90.000,E1 99.095} C_DIS
LIN {X 0.177,Y -481.411,Z 1254.548,A 0.000,B 0.000,C 90.000,E1 98.568} C_DIS
LIN {X -0.135,Y -481.173,Z 1254.545,A 0.000,B 0.000,C 90.000,E1 98.106} C_DIS
LIN {X 0.035,Y -479.922,Z 1254.542,A 0.000,B 0.000,C 90.000,E1 97.587} C_DIS
LIN {X -0.088,Y -478.857,Z 1254.541,A 0.000,B 0.000,C 90.000,E1 97.352} C_DIS
LIN {X 0.203,Y -477.427,Z 1254.539,A 0.000,B 0.000,C 90.000,E1 97.068} C_DIS
LIN {X -0.154,Y -455.590,Z 1254.523,A 0.000,B 0.000,C 90.000,E1 94.073} C_DIS
LIN {X 0.051,Y -435.165,Z 1254.505,A 0.000,B 0.000,C 90.000,E1 90.917} C_DIS
LIN {X -0.142,Y -418.434,Z 1254.489,A 0.000,B 0.000,C 90.000,E1 87.993} C_DIS
LIN {X 0.108,Y -408.446,Z 1254.478,A 0.000,B 0.000,C 90.000,E1 86.045} C_DIS
LIN {X 0.185,Y -398.361,Z 1254.467,A 0.000,B 0.000,C 90.000,E1 84.090} C_DIS
LIN {X 0.097,Y -388.105,Z 1254.456,A 0.000,B 0.000,C 90.000,E1 82.129} C_DIS
LIN {X -0.111,Y -379.162,Z 1254.447,A 0.000,B 0.000,C 90.000,E1 80.443} C_DIS
LIN {X -0.103,Y -369.921,Z 1254.437,A 0.000,B 0.000,C 90.000,E1 78.701} C_DIS
LIN {X -0.116,Y -360.327,Z 1254.427,A 0.000,B 0.000,C 90.000,E1 76.937} C_DIS
LIN {X 0.065,Y -348.922,Z 1254.416,A 0.000,B 0.000,C 90.000,E1 74.810} C_DIS
LIN {X 0.086,Y -337.516,Z 1254.404,A 0.000,B 0.000,C 90.000,E1 72.670} C_DIS
LIN {X -0.022,Y -323.247,Z 1254.388,A 0.000,B 0.000,C 90.000,E1 69.880} C_DIS
LIN {X -0.036,Y -306.880,Z 1254.369,A 0.000,B 0.000,C 90.000,E1 66.357} C_DIS
LIN {X -0.096,Y -292.158,Z 1254.349,A 0.000,B 0.000,C 90.000,E1 62.743} C_DIS
LIN {X 0.070,Y -280.172,Z 1254.330,A 0.000,B 0.000,C 90.000,E1 59.331} C_DIS
LIN {X 0.132,Y -270.287,Z 1254.313,A 0.000,B 0.000,C 90.000,E1 56.215} C_DIS
LIN {X 0.067,Y -260.217,Z 1254.293,A 0.000,B 0.000,C 90.000,E1 52.718} C_DIS
LIN {X 0.076,Y -251.038,Z 1254.273,A 0.000,B 0.000,C 90.000,E1 49.138} C_DIS
LIN {X 0.112,Y -242.405,Z 1254.253,A 0.000,B 0.000,C 90.000,E1 45.486} C_DIS
LIN {X 0.106,Y -235.904,Z 1254.236,A 0.000,B 0.000,C 90.000,E1 42.528} C_DIS
LIN {X -0.120,Y -228.062,Z 1254.216,A 0.000,B 0.000,C 90.000,E1 38.830} C_DIS
LIN {X 0.029,Y -220.838,Z 1254.194,A 0.000,B 0.000,C 90.000,E1 34.978} C_DIS
LIN {X -0.062,Y -214.263,Z 1254.173,A 0.000,B 0.000,C 90.000,E1 31.131} C_DIS
LIN {X -0.060,Y -208.494,Z 1254.151,A 0.000,B 0.000,C 90.000,E1 27.206} C_DIS
LIN {X 0.041,Y -203.625,Z 1254.129,A 0.000,B 0.000,C 90.000,E1 23.206} C_DIS
LIN {X -0.066,Y -198.770,Z 1254.102,A 0.000,B 0.000,C 90.000,E1 18.417} C_DIS
LIN {X -0.025,Y -195.003,Z 1254.075,A 0.000,B 0.000,C 90.000,E1 13.536} C_DIS
LIN {X -0.043,Y -192.195,Z 1254.043,A 0.000,B 0.000,C 90.000,E1 7.814} C_DIS
LIN {X -0.075,Y -193.392,Z 1253.965,A 0.000,B 0.000,C 90.000,E1 353.799} C_DIS
LIN {X 0.010,Y -196.833,Z 1253.934,A 0.000,B 0.000,C 90.000,E1 348.049} C_DIS
LIN {X -0.044,Y -200.980,Z 1253.907,A 0.000,B 0.000,C 90.000,E1 343.196} C_DIS
LIN {X 0.023,Y -205.197,Z 1253.884,A 0.000,B 0.000,C 90.000,E1 339.156} C_DIS
LIN {X 0.008,Y -210.188,Z 1253.862,A 0.000,B 0.000,C 90.000,E1 335.177} C_DIS
LIN {X -0.066,Y -215.753,Z 1253.840,A 0.000,B 0.000,C 90.000,E1 331.257} C_DIS
LIN {X 0.080,Y -222.072,Z 1253.819,A 0.000,B 0.000,C 90.000,E1 327.327} C_DIS
LIN {X 0.044,Y -229.060,Z 1253.797,A 0.000,B 0.000,C 90.000,E1 323.497} C_DIS
LIN {X -0.089,Y -236.876,Z 1253.776,A 0.000,B 0.000,C 90.000,E1 319.747} C_DIS
LIN {X 0.135,Y -245.626,Z 1253.756,A 0.000,B 0.000,C 90.000,E1 315.972} C_DIS
LIN {X 0.107,Y -254.576,Z 1253.737,A 0.000,B 0.000,C 90.000,E1 312.690} C_DIS
LIN {X 0.078,Y -261.408,Z 1253.725,A 0.000,B 0.000,C 90.000,E1 310.539} C_DIS
LIN {X -0.166,Y -269.103,Z 1253.714,A 0.000,B 0.000,C 90.000,E1 308.463} C_DIS
LIN {X 0.068,Y -276.296,Z 1253.704,A 0.000,B 0.000,C 90.000,E1 306.664} C_DIS
LIN {X -0.046,Y -287.566,Z 1253.690,A 0.000,B 0.000,C 90.000,E1 304.278} C_DIS
LIN {X -0.081,Y -298.211,Z 1253.679,A 0.000,B 0.000,C 90.000,E1 302.260} C_DIS
LIN {X -0.016,Y -308.098,Z 1253.670,A 0.000,B 0.000,C 90.000,E1 300.590} C_DIS
LIN {X 0.067,Y -319.291,Z 1253.661,A 0.000,B 0.000,C 90.000,E1 298.949} C_DIS
LIN {X 0.054,Y -341.618,Z 1253.645,A 0.000,B 0.000,C 90.000,E1 296.104} C_DIS
LIN {X -0.067,Y -357.116,Z 1253.635,A 0.000,B 0.000,C 90.000,E1 294.335} C_DIS
LIN {X -0.165,Y -370.043,Z 1253.627,A 0.000,B 0.000,C 90.000,E1 292.898} C_DIS
LIN {X -0.150,Y -382.848,Z 1253.619,A 0.000,B 0.000,C 90.000,E1 291.461} C_DIS
LIN {X -0.004,Y -400.874,Z 1253.608,A 0.000,B 0.000,C 90.000,E1 289.450} C_DIS
LIN {X 0.130,Y -416.146,Z 1253.599,A 0.000,B 0.000,C 90.000,E1 287.819} C_DIS
LIN {X -0.075,Y -423.570,Z 1253.595,A 0.000,B 0.000,C 90.000,E1 287.040} C_DIS
LIN {X -0.045,Y -432.888,Z 1253.589,A 0.000,B 0.000,C 90.000,E1 285.953} C_DIS
LIN {X 0.086,Y -439.234,Z 1253.584,A 0.000,B 0.000,C 90.000,E1 285.134} C_DIS
LIN {X -0.037,Y -444.975,Z 1253.580,A 0.000,B 0.000,C 90.000,E1 284.356} C_DIS
LIN {X -0.221,Y -450.012,Z 1253.575,A 0.000,B 0.000,C 90.000,E1 283.592} C_DIS
LIN {X 0.079,Y -454.411,Z 1253.571,A 0.000,B 0.000,C 90.000,E1 282.771} C_DIS
LIN {X -0.018,Y -458.108,Z 1253.567,A 0.000,B 0.000,C 90.000,E1 282.007} C_DIS
LIN {X -0.090,Y -461.142,Z 1253.562,A 0.000,B 0.000,C 90.000,E1 281.243} C_DIS
LIN {X 0.022,Y -462.843,Z 1253.560,A 0.000,B 0.000,C 90.000,E1 280.715} C_DIS
LIN {X 0.061,Y -464.302,Z 1253.557,A 0.000,B 0.000,C 90.000,E1 280.197} C_DIS
LIN {X 0.194,Y -465.442,Z 1253.554,A 0.000,B 0.000,C 90.000,E1 279.670} C_DIS
LIN {X -0.203,Y -466.336,Z 1253.551,A 0.000,B 0.000,C 90.000,E1 279.208} C_DIS
LIN {X -0.060,Y -466.914,Z 1253.548,A 0.000,B 0.000,C 90.000,E1 278.681} C_DIS
LIN {X 0.016,Y -467.166,Z 1253.545,A 0.000,B 0.000,C 90.000,E1 278.163} C_DIS
LIN {X 0.099,Y -466.983,Z 1253.542,A 0.000,B 0.000,C 90.000,E1 277.644} C_DIS
LIN {X 0.184,Y -466.396,Z 1253.540,A 0.000,B 0.000,C 90.000,E1 277.125} C_DIS
LIN {X -0.194,Y -465.372,Z 1253.537,A 0.000,B 0.000,C 90.000,E1 276.663} C_DIS
LIN {X -0.111,Y -463.914,Z 1253.534,A 0.000,B 0.000,C 90.000,E1 276.144} C_DIS
LIN {X -0.035,Y -462.099,Z 1253.531,A 0.000,B 0.000,C 90.000,E1 275.625} C_DIS
LIN {X -0.194,Y -458.580,Z 1253.527,A 0.000,B 0.000,C 90.000,E1 274.878} C_DIS
LIN {X -0.152,Y -455.682,Z 1253.524,A 0.000,B 0.000,C 90.000,E1 274.359} C_DIS
LIN {X 0.075,Y -454.008,Z 1253.523,A 0.000,B 0.000,C 90.000,E1 274.073} C_DIS
LIN {X 0.089,Y -449.881,Z 1253.520,A 0.000,B 0.000,C 90.000,E1 273.555} C_DIS
LIN {X -0.151,Y -447.442,Z 1253.518,A 0.000,B 0.000,C 90.000,E1 273.326} C_DIS
LIN {X -0.012,Y -441.750,Z 1253.516,A 0.000,B 0.000,C 90.000,E1 272.808} C_DIS
LIN {X 0.079,Y -435.366,Z 1253.513,A 0.000,B 0.000,C 90.000,E1 272.350} C_DIS
LIN {X -0.158,Y -428.531,Z 1253.511,A 0.000,B 0.000,C 90.000,E1 272.007} C_DIS
LIN {X 0.092,Y -421.571,Z 1253.509,A 0.000,B 0.000,C 90.000,E1 271.661} C_DIS
LIN {X -0.141,Y -414.493,Z 1253.508,A 0.000,B 0.000,C 90.000,E1 271.432} C_DIS
LIN {X 0.049,Y -403.711,Z 1253.506,A 0.000,B 0.000,C 90.000,E1 271.088} C_DIS
LIN {X -0.029,Y -392.601,Z 1253.505,A 0.000,B 0.000,C 90.000,E1 270.859} C_DIS
LIN {X -0.087,Y -384.300,Z 1253.504,A 0.000,B 0.000,C 90.000,E1 270.745} C_DIS
LIN {X -0.112,Y -371.016,Z 1253.503,A 0.000,B 0.000,C 90.000,E1 270.630} C_DIS
LIN {X 0.119,Y -364.624,Z 1253.503,A 0.000,B 0.000,C 90.000,E1 270.573} C_DIS
LIN {X 0.038,Y -181.551,Z 1253.503,A 0.000,B 0.000,C 90.000,E1 270.573} C_DIS
LIN {X -0.004,Y -181.286,Z 1253.494,A 0.000,B 0.000,C 90.000,E1 268.854} C_DIS
LIN {X 0.045,Y -180.907,Z 1253.475,A 0.000,B 0.000,C 90.000,E1 265.469} C_DIS
LIN {X -0.079,Y -180.743,Z 1253.470,A 0.000,B 0.000,C 90.000,E1 264.666} C_DIS
LIN {X 0.023,Y -178.834,Z 1253.442,A 0.000,B 0.000,C 90.000,E1 259.567} C_DIS
LIN {X 0.056,Y -175.878,Z 1253.414,A 0.000,B 0.000,C 90.000,E1 254.464} C_DIS
LIN {X -0.007,Y -174.538,Z 1253.404,A 0.000,B 0.000,C 90.000,E1 252.779} C_DIS
LIN {X 0.086,Y -171.522,Z 1253.380,A 0.000,B 0.000,C 90.000,E1 248.465} C_DIS
LIN {X 0.072,Y -167.749,Z 1253.357,A 0.000,B 0.000,C 90.000,E1 244.152} C_DIS
LIN {X 0.010,Y -166.451,Z 1253.347,A 0.000,B 0.000,C 90.000,E1 242.436} C_DIS
LIN {X 0.001,Y -163.167,Z 1253.328,A 0.000,B 0.000,C 90.000,E1 238.948} C_DIS
LIN {X 0.049,Y -161.127,Z 1253.313,A 0.000,B 0.000,C 90.000,E1 236.294} C_DIS
LIN {X -0.047,Y -157.148,Z 1253.288,A 0.000,B 0.000,C 90.000,E1 231.904} C_DIS
LIN {X -0.024,Y -155.881,Z 1253.278,A 0.000,B 0.000,C 90.000,E1 230.114} C_DIS
LIN {X -0.066,Y -152.131,Z 1253.253,A 0.000,B 0.000,C 90.000,E1 225.648} C_DIS
LIN {X -0.046,Y -150.381,Z 1253.238,A 0.000,B 0.000,C 90.000,E1 222.933} C_DIS
LIN {X -0.021,Y -147.113,Z 1253.213,A 0.000,B 0.000,C 90.000,E1 218.382} C_DIS
LIN {X -0.030,Y -145.679,Z 1253.198,A 0.000,B 0.000,C 90.000,E1 215.644} C_DIS
LIN {X -0.031,Y -143.062,Z 1253.172,A 0.000,B 0.000,C 90.000,E1 211.052} C_DIS
LIN {X 0.026,Y -141.684,Z 1253.152,A 0.000,B 0.000,C 90.000,E1 207.334} C_DIS
LIN {X 0.004,Y -139.458,Z 1253.116,A 0.000,B 0.000,C 90.000,E1 200.844} C_DIS
LIN {X 0.055,Y -139.192,Z 1253.105,A 0.000,B 0.000,C 90.000,E1 198.960} C_DIS
